						10:	(*Consigne epaisseur pour la nouvelle vitesse*)
							VAR_ParameterWriter.fbClientDataExcha.txBuffer[0]:=16#08;
							VAR_ParameterWriter.fbClientDataExcha.txBuffer[1]:=16#00;
							VAR_ParameterWriter.fbClientDataExcha.txBuffer[2]:= F_ToASC('U');
							VAR_ParameterWriter.fbClientDataExcha.txBuffer[3]:= F_ToASC('F');
							VAR_ParameterWriter.fbClientDataExcha.txBuffer[4]:= 16#0A;
							VAR_ParameterWriter.fbClientDataExcha.txBuffer[5]:= 16#01;
							MEMCPY(ADR(VAR_ParameterWriter.fbClientDataExcha.txBuffer[6]),ADR(I_Thick_SP),4);
							VAR_ParameterWriter.fbClientDataExcha.txBuffer[10] := VAR_ParameterWriter.fbClientDataExcha.txBuffer[2] +
												VAR_ParameterWriter.fbClientDataExcha.txBuffer[3] +
												VAR_ParameterWriter.fbClientDataExcha.txBuffer[4] +
												VAR_ParameterWriter.fbClientDataExcha.txBuffer[5] +
												VAR_ParameterWriter.fbClientDataExcha.txBuffer[6] +
												VAR_ParameterWriter.fbClientDataExcha.txBuffer[7] +
												VAR_ParameterWriter.fbClientDataExcha.txBuffer[8] +
												VAR_ParameterWriter.fbClientDataExcha.txBuffer[9];
							VAR_ParameterWriter.fbClientDataExcha.nbTransmittedChar := 11;
							VAR_ParameterWriter.fbClientDataExcha.nbExpectedChar := 6;


						11:	(*Nouvelle consigne de vitesse*)
							VAR_ParameterWriter.fbClientDataExcha.txBuffer[0]:=16#08;
							VAR_ParameterWriter.fbClientDataExcha.txBuffer[1]:=16#00;
							VAR_ParameterWriter.fbClientDataExcha.txBuffer[2]:= F_ToASC('U');
							VAR_ParameterWriter.fbClientDataExcha.txBuffer[3]:= F_ToASC('F');
							VAR_ParameterWriter.fbClientDataExcha.txBuffer[4]:= 16#0B;
							VAR_ParameterWriter.fbClientDataExcha.txBuffer[5]:= 16#01;
							MEMCPY(ADR(VAR_ParameterWriter.fbClientDataExcha.txBuffer[6]),ADR(I_New_Rate),4);
							VAR_ParameterWriter.fbClientDataExcha.txBuffer[10] := VAR_ParameterWriter.fbClientDataExcha.txBuffer[2] +
												VAR_ParameterWriter.fbClientDataExcha.txBuffer[3] +
												VAR_ParameterWriter.fbClientDataExcha.txBuffer[4] +
												VAR_ParameterWriter.fbClientDataExcha.txBuffer[5] +
												VAR_ParameterWriter.fbClientDataExcha.txBuffer[6] +
												VAR_ParameterWriter.fbClientDataExcha.txBuffer[7] +
												VAR_ParameterWriter.fbClientDataExcha.txBuffer[8] +
												VAR_ParameterWriter.fbClientDataExcha.txBuffer[9];
							VAR_ParameterWriter.fbClientDataExcha.nbTransmittedChar := 11;
							VAR_ParameterWriter.fbClientDataExcha.nbExpectedChar := 6;


						12:	(*Temps de monté à la nouvelle vitesse*)
							VAR_ParameterWriter.fbClientDataExcha.txBuffer[0]:=16#08;
							VAR_ParameterWriter.fbClientDataExcha.txBuffer[1]:=16#00;
							VAR_ParameterWriter.fbClientDataExcha.txBuffer[2]:= F_ToASC('U');
							VAR_ParameterWriter.fbClientDataExcha.txBuffer[3]:= F_ToASC('F');
							VAR_ParameterWriter.fbClientDataExcha.txBuffer[4]:= 16#0C;
							VAR_ParameterWriter.fbClientDataExcha.txBuffer[5]:= 16#01;
							TEMP_DWORD := UINT_TO_DWORD(I_Rate_Ramp_Time);
							MEMCPY(ADR(VAR_ParameterWriter.fbClientDataExcha.txBuffer[6]),ADR(TEMP_DWORD),4);
							VAR_ParameterWriter.fbClientDataExcha.txBuffer[10] := VAR_ParameterWriter.fbClientDataExcha.txBuffer[2] +
												VAR_ParameterWriter.fbClientDataExcha.txBuffer[3] +
												VAR_ParameterWriter.fbClientDataExcha.txBuffer[4] +
												VAR_ParameterWriter.fbClientDataExcha.txBuffer[5] +
												VAR_ParameterWriter.fbClientDataExcha.txBuffer[6] +
												VAR_ParameterWriter.fbClientDataExcha.txBuffer[7] +
												VAR_ParameterWriter.fbClientDataExcha.txBuffer[8] +
												VAR_ParameterWriter.fbClientDataExcha.txBuffer[9];
							VAR_ParameterWriter.fbClientDataExcha.nbTransmittedChar := 11;
							VAR_ParameterWriter.fbClientDataExcha.nbExpectedChar := 6;


						13:	(*Rate Watcher Accuracy*)
							VAR_ParameterWriter.fbClientDataExcha.txBuffer[0]:=16#08;
							VAR_ParameterWriter.fbClientDataExcha.txBuffer[1]:=16#00;
							VAR_ParameterWriter.fbClientDataExcha.txBuffer[2]:= F_ToASC('U');
							VAR_ParameterWriter.fbClientDataExcha.txBuffer[3]:= F_ToASC('F');
							VAR_ParameterWriter.fbClientDataExcha.txBuffer[4]:= 16#0D;
							VAR_ParameterWriter.fbClientDataExcha.txBuffer[5]:= 16#01;
							TEMP_DWORD := INT_TO_DWORD(I_Rate_Watcher_Accuracy);
							MEMCPY(ADR(VAR_ParameterWriter.fbClientDataExcha.txBuffer[6]),ADR(TEMP_DWORD),4);
							VAR_ParameterWriter.fbClientDataExcha.txBuffer[10] := VAR_ParameterWriter.fbClientDataExcha.txBuffer[2] +
												VAR_ParameterWriter.fbClientDataExcha.txBuffer[3] +
												VAR_ParameterWriter.fbClientDataExcha.txBuffer[4] +
												VAR_ParameterWriter.fbClientDataExcha.txBuffer[5] +
												VAR_ParameterWriter.fbClientDataExcha.txBuffer[6] +
												VAR_ParameterWriter.fbClientDataExcha.txBuffer[7] +
												VAR_ParameterWriter.fbClientDataExcha.txBuffer[8] +
												VAR_ParameterWriter.fbClientDataExcha.txBuffer[9];
							VAR_ParameterWriter.fbClientDataExcha.nbTransmittedChar := 11;
							VAR_ParameterWriter.fbClientDataExcha.nbExpectedChar := 6;


						14:	(*RW hold time*)
							VAR_ParameterWriter.fbClientDataExcha.txBuffer[0]:=16#08;
							VAR_ParameterWriter.fbClientDataExcha.txBuffer[1]:=16#00;
							VAR_ParameterWriter.fbClientDataExcha.txBuffer[2]:= F_ToASC('U');
							VAR_ParameterWriter.fbClientDataExcha.txBuffer[3]:= F_ToASC('F');
							VAR_ParameterWriter.fbClientDataExcha.txBuffer[4]:= 16#0E;
							VAR_ParameterWriter.fbClientDataExcha.txBuffer[5]:= 16#01;
							TEMP_DWORD := INT_TO_DWORD(I_RW_Hold_Time);
							MEMCPY(ADR(VAR_ParameterWriter.fbClientDataExcha.txBuffer[6]),ADR(TEMP_DWORD),4);
							VAR_ParameterWriter.fbClientDataExcha.txBuffer[10] := VAR_ParameterWriter.fbClientDataExcha.txBuffer[2] +
												VAR_ParameterWriter.fbClientDataExcha.txBuffer[3] +
												VAR_ParameterWriter.fbClientDataExcha.txBuffer[4] +
												VAR_ParameterWriter.fbClientDataExcha.txBuffer[5] +
												VAR_ParameterWriter.fbClientDataExcha.txBuffer[6] +
												VAR_ParameterWriter.fbClientDataExcha.txBuffer[7] +
												VAR_ParameterWriter.fbClientDataExcha.txBuffer[8] +
												VAR_ParameterWriter.fbClientDataExcha.txBuffer[9];
							VAR_ParameterWriter.fbClientDataExcha.nbTransmittedChar := 11;
							VAR_ParameterWriter.fbClientDataExcha.nbExpectedChar := 6;


						15:	(*Sensor à utiliser*)
							VAR_ParameterWriter.fbClientDataExcha.txBuffer[0]:=16#08;
							VAR_ParameterWriter.fbClientDataExcha.txBuffer[1]:=16#00;
							VAR_ParameterWriter.fbClientDataExcha.txBuffer[2]:= F_ToASC('U');
							VAR_ParameterWriter.fbClientDataExcha.txBuffer[3]:= F_ToASC('F');
							VAR_ParameterWriter.fbClientDataExcha.txBuffer[4]:= 16#0F;
							VAR_ParameterWriter.fbClientDataExcha.txBuffer[5]:= 16#01;
							TEMP_DWORD := BYTE_TO_DWORD(I_Sensor);
							MEMCPY(ADR(VAR_ParameterWriter.fbClientDataExcha.txBuffer[6]),ADR(TEMP_DWORD),4);
							VAR_ParameterWriter.fbClientDataExcha.txBuffer[10] := VAR_ParameterWriter.fbClientDataExcha.txBuffer[2] +
												VAR_ParameterWriter.fbClientDataExcha.txBuffer[3] +
												VAR_ParameterWriter.fbClientDataExcha.txBuffer[4] +
												VAR_ParameterWriter.fbClientDataExcha.txBuffer[5] +
												VAR_ParameterWriter.fbClientDataExcha.txBuffer[6] +
												VAR_ParameterWriter.fbClientDataExcha.txBuffer[7] +
												VAR_ParameterWriter.fbClientDataExcha.txBuffer[8] +
												VAR_ParameterWriter.fbClientDataExcha.txBuffer[9];
							VAR_ParameterWriter.fbClientDataExcha.nbTransmittedChar := 11;
							VAR_ParameterWriter.fbClientDataExcha.nbExpectedChar := 6;


						16:	(*Facteur de correction 1*)
							VAR_ParameterWriter.fbClientDataExcha.txBuffer[0]:=16#08;
							VAR_ParameterWriter.fbClientDataExcha.txBuffer[1]:=16#00;
							VAR_ParameterWriter.fbClientDataExcha.txBuffer[2]:= F_ToASC('U');
							VAR_ParameterWriter.fbClientDataExcha.txBuffer[3]:= F_ToASC('F');
							VAR_ParameterWriter.fbClientDataExcha.txBuffer[4]:= 16#10;
							VAR_ParameterWriter.fbClientDataExcha.txBuffer[5]:= 16#01;
							MEMCPY(ADR(VAR_ParameterWriter.fbClientDataExcha.txBuffer[6]),ADR(I_Tool_Factor1),4);
							VAR_ParameterWriter.fbClientDataExcha.txBuffer[10] := VAR_ParameterWriter.fbClientDataExcha.txBuffer[2] +
												VAR_ParameterWriter.fbClientDataExcha.txBuffer[3] +
												VAR_ParameterWriter.fbClientDataExcha.txBuffer[4] +
												VAR_ParameterWriter.fbClientDataExcha.txBuffer[5] +
												VAR_ParameterWriter.fbClientDataExcha.txBuffer[6] +
												VAR_ParameterWriter.fbClientDataExcha.txBuffer[7] +
												VAR_ParameterWriter.fbClientDataExcha.txBuffer[8] +
												VAR_ParameterWriter.fbClientDataExcha.txBuffer[9];
							VAR_ParameterWriter.fbClientDataExcha.nbTransmittedChar := 11;
							VAR_ParameterWriter.fbClientDataExcha.nbExpectedChar := 6;



						17:	(*Facteur de correction 2*)
							VAR_ParameterWriter.fbClientDataExcha.txBuffer[0]:=16#08;
							VAR_ParameterWriter.fbClientDataExcha.txBuffer[1]:=16#00;
							VAR_ParameterWriter.fbClientDataExcha.txBuffer[2]:= F_ToASC('U');
							VAR_ParameterWriter.fbClientDataExcha.txBuffer[3]:= F_ToASC('F');
							VAR_ParameterWriter.fbClientDataExcha.txBuffer[4]:= 16#11;
							VAR_ParameterWriter.fbClientDataExcha.txBuffer[5]:= 16#01;
							MEMCPY(ADR(VAR_ParameterWriter.fbClientDataExcha.txBuffer[6]),ADR(I_Tool_Factor2),4);
							VAR_ParameterWriter.fbClientDataExcha.txBuffer[10] := VAR_ParameterWriter.fbClientDataExcha.txBuffer[2] +
												VAR_ParameterWriter.fbClientDataExcha.txBuffer[3] +
												VAR_ParameterWriter.fbClientDataExcha.txBuffer[4] +
												VAR_ParameterWriter.fbClientDataExcha.txBuffer[5] +
												VAR_ParameterWriter.fbClientDataExcha.txBuffer[6] +
												VAR_ParameterWriter.fbClientDataExcha.txBuffer[7] +
												VAR_ParameterWriter.fbClientDataExcha.txBuffer[8] +
												VAR_ParameterWriter.fbClientDataExcha.txBuffer[9];
							VAR_ParameterWriter.fbClientDataExcha.nbTransmittedChar := 11;
							VAR_ParameterWriter.fbClientDataExcha.nbExpectedChar := 6;



						18:	(*Xtal stabilility single*)
							VAR_ParameterWriter.fbClientDataExcha.txBuffer[0]:=16#08;
							VAR_ParameterWriter.fbClientDataExcha.txBuffer[1]:=16#00;
							VAR_ParameterWriter.fbClientDataExcha.txBuffer[2]:= F_ToASC('U');
							VAR_ParameterWriter.fbClientDataExcha.txBuffer[3]:= F_ToASC('F');
							VAR_ParameterWriter.fbClientDataExcha.txBuffer[4]:= 16#12;
							VAR_ParameterWriter.fbClientDataExcha.txBuffer[5]:= 16#01;
							TEMP_DWORD := UINT_TO_DWORD(I_Stab_Single);
							MEMCPY(ADR(VAR_ParameterWriter.fbClientDataExcha.txBuffer[6]),ADR(TEMP_DWORD),4);
							VAR_ParameterWriter.fbClientDataExcha.txBuffer[10] := VAR_ParameterWriter.fbClientDataExcha.txBuffer[2] +
												VAR_ParameterWriter.fbClientDataExcha.txBuffer[3] +
												VAR_ParameterWriter.fbClientDataExcha.txBuffer[4] +
												VAR_ParameterWriter.fbClientDataExcha.txBuffer[5] +
												VAR_ParameterWriter.fbClientDataExcha.txBuffer[6] +
												VAR_ParameterWriter.fbClientDataExcha.txBuffer[7] +
												VAR_ParameterWriter.fbClientDataExcha.txBuffer[8] +
												VAR_ParameterWriter.fbClientDataExcha.txBuffer[9];
							VAR_ParameterWriter.fbClientDataExcha.nbTransmittedChar := 11;
							VAR_ParameterWriter.fbClientDataExcha.nbExpectedChar := 6;


						19:	(*Xtal stabilility total*)
							VAR_ParameterWriter.fbClientDataExcha.txBuffer[0]:=16#08;
							VAR_ParameterWriter.fbClientDataExcha.txBuffer[1]:=16#00;
							VAR_ParameterWriter.fbClientDataExcha.txBuffer[2]:= F_ToASC('U');
							VAR_ParameterWriter.fbClientDataExcha.txBuffer[3]:= F_ToASC('F');
							VAR_ParameterWriter.fbClientDataExcha.txBuffer[4]:= 16#13;
							VAR_ParameterWriter.fbClientDataExcha.txBuffer[5]:= 16#01;
							TEMP_DWORD := UINT_TO_DWORD(I_Stab_Total);
							MEMCPY(ADR(VAR_ParameterWriter.fbClientDataExcha.txBuffer[6]),ADR(TEMP_DWORD),4);
							VAR_ParameterWriter.fbClientDataExcha.txBuffer[10] := VAR_ParameterWriter.fbClientDataExcha.txBuffer[2] +
												VAR_ParameterWriter.fbClientDataExcha.txBuffer[3] +
												VAR_ParameterWriter.fbClientDataExcha.txBuffer[4] +
												VAR_ParameterWriter.fbClientDataExcha.txBuffer[5] +
												VAR_ParameterWriter.fbClientDataExcha.txBuffer[6] +
												VAR_ParameterWriter.fbClientDataExcha.txBuffer[7] +
												VAR_ParameterWriter.fbClientDataExcha.txBuffer[8] +
												VAR_ParameterWriter.fbClientDataExcha.txBuffer[9];
							VAR_ParameterWriter.fbClientDataExcha.nbTransmittedChar := 11;
							VAR_ParameterWriter.fbClientDataExcha.nbExpectedChar := 6;


						20:	(*Xtal quality percent*)
							VAR_ParameterWriter.fbClientDataExcha.txBuffer[0]:=16#08;
							VAR_ParameterWriter.fbClientDataExcha.txBuffer[1]:=16#00;
							VAR_ParameterWriter.fbClientDataExcha.txBuffer[2]:= F_ToASC('U');
							VAR_ParameterWriter.fbClientDataExcha.txBuffer[3]:= F_ToASC('F');
							VAR_ParameterWriter.fbClientDataExcha.txBuffer[4]:= 16#14;
							VAR_ParameterWriter.fbClientDataExcha.txBuffer[5]:= 16#01;
							TEMP_DWORD := USINT_TO_DWORD(I_Quality_percent);
							MEMCPY(ADR(VAR_ParameterWriter.fbClientDataExcha.txBuffer[6]),ADR(TEMP_DWORD),4);
							VAR_ParameterWriter.fbClientDataExcha.txBuffer[10] := VAR_ParameterWriter.fbClientDataExcha.txBuffer[2] +
												VAR_ParameterWriter.fbClientDataExcha.txBuffer[3] +
												VAR_ParameterWriter.fbClientDataExcha.txBuffer[4] +
												VAR_ParameterWriter.fbClientDataExcha.txBuffer[5] +
												VAR_ParameterWriter.fbClientDataExcha.txBuffer[6] +
												VAR_ParameterWriter.fbClientDataExcha.txBuffer[7] +
												VAR_ParameterWriter.fbClientDataExcha.txBuffer[8] +
												VAR_ParameterWriter.fbClientDataExcha.txBuffer[9];
							VAR_ParameterWriter.fbClientDataExcha.nbTransmittedChar := 11;
							VAR_ParameterWriter.fbClientDataExcha.nbExpectedChar := 6;


						21:	(*Xtal quality Counts*)
							VAR_ParameterWriter.fbClientDataExcha.txBuffer[0]:=16#08;
							VAR_ParameterWriter.fbClientDataExcha.txBuffer[1]:=16#00;
							VAR_ParameterWriter.fbClientDataExcha.txBuffer[2]:= F_ToASC('U');
							VAR_ParameterWriter.fbClientDataExcha.txBuffer[3]:= F_ToASC('F');
							VAR_ParameterWriter.fbClientDataExcha.txBuffer[4]:= 16#15;
							VAR_ParameterWriter.fbClientDataExcha.txBuffer[5]:= 16#01;
							TEMP_DWORD := USINT_TO_DWORD(I_Quality_Counts);
							MEMCPY(ADR(VAR_ParameterWriter.fbClientDataExcha.txBuffer[6]),ADR(TEMP_DWORD),4);
							VAR_ParameterWriter.fbClientDataExcha.txBuffer[10] := VAR_ParameterWriter.fbClientDataExcha.txBuffer[2] +
												VAR_ParameterWriter.fbClientDataExcha.txBuffer[3] +
												VAR_ParameterWriter.fbClientDataExcha.txBuffer[4] +
												VAR_ParameterWriter.fbClientDataExcha.txBuffer[5] +
												VAR_ParameterWriter.fbClientDataExcha.txBuffer[6] +
												VAR_ParameterWriter.fbClientDataExcha.txBuffer[7] +
												VAR_ParameterWriter.fbClientDataExcha.txBuffer[8] +
												VAR_ParameterWriter.fbClientDataExcha.txBuffer[9];
							VAR_ParameterWriter.fbClientDataExcha.nbTransmittedChar := 11;
							VAR_ParameterWriter.fbClientDataExcha.nbExpectedChar := 6;


						22:	(*Source*)
							VAR_ParameterWriter.fbClientDataExcha.txBuffer[0]:=16#08;
							VAR_ParameterWriter.fbClientDataExcha.txBuffer[1]:=16#00;
							VAR_ParameterWriter.fbClientDataExcha.txBuffer[2]:= F_ToASC('U');
							VAR_ParameterWriter.fbClientDataExcha.txBuffer[3]:= F_ToASC('F');
							VAR_ParameterWriter.fbClientDataExcha.txBuffer[4]:= 16#16;
							VAR_ParameterWriter.fbClientDataExcha.txBuffer[5]:= 16#01;
							TEMP_DWORD := BYTE_TO_DWORD(I_Source);
							MEMCPY(ADR(VAR_ParameterWriter.fbClientDataExcha.txBuffer[6]),ADR(TEMP_DWORD),4);
							VAR_ParameterWriter.fbClientDataExcha.txBuffer[10] := VAR_ParameterWriter.fbClientDataExcha.txBuffer[2] +
												VAR_ParameterWriter.fbClientDataExcha.txBuffer[3] +
												VAR_ParameterWriter.fbClientDataExcha.txBuffer[4] +
												VAR_ParameterWriter.fbClientDataExcha.txBuffer[5] +
												VAR_ParameterWriter.fbClientDataExcha.txBuffer[6] +
												VAR_ParameterWriter.fbClientDataExcha.txBuffer[7] +
												VAR_ParameterWriter.fbClientDataExcha.txBuffer[8] +
												VAR_ParameterWriter.fbClientDataExcha.txBuffer[9];
							VAR_ParameterWriter.fbClientDataExcha.nbTransmittedChar := 11;
							VAR_ParameterWriter.fbClientDataExcha.nbExpectedChar := 6;


						23:	(*Source*)
							VAR_ParameterWriter.fbClientDataExcha.txBuffer[0]:=16#08;
							VAR_ParameterWriter.fbClientDataExcha.txBuffer[1]:=16#00;
							VAR_ParameterWriter.fbClientDataExcha.txBuffer[2]:= F_ToASC('U');
							VAR_ParameterWriter.fbClientDataExcha.txBuffer[3]:= F_ToASC('F');
							VAR_ParameterWriter.fbClientDataExcha.txBuffer[4]:= 16#17;
							VAR_ParameterWriter.fbClientDataExcha.txBuffer[5]:= 16#01;
							TEMP_DWORD := BYTE_TO_DWORD(I_Crucible_Nb);
							MEMCPY(ADR(VAR_ParameterWriter.fbClientDataExcha.txBuffer[6]),ADR(TEMP_DWORD),4);
							VAR_ParameterWriter.fbClientDataExcha.txBuffer[10] := VAR_ParameterWriter.fbClientDataExcha.txBuffer[2] +
												VAR_ParameterWriter.fbClientDataExcha.txBuffer[3] +
												VAR_ParameterWriter.fbClientDataExcha.txBuffer[4] +
												VAR_ParameterWriter.fbClientDataExcha.txBuffer[5] +
												VAR_ParameterWriter.fbClientDataExcha.txBuffer[6] +
												VAR_ParameterWriter.fbClientDataExcha.txBuffer[7] +
												VAR_ParameterWriter.fbClientDataExcha.txBuffer[8] +
												VAR_ParameterWriter.fbClientDataExcha.txBuffer[9];
							VAR_ParameterWriter.fbClientDataExcha.nbTransmittedChar := 11;
							VAR_ParameterWriter.fbClientDataExcha.nbExpectedChar := 6;


						24:	(*PID Gain*)
							VAR_ParameterWriter.fbClientDataExcha.txBuffer[0]:=16#08;
							VAR_ParameterWriter.fbClientDataExcha.txBuffer[1]:=16#00;
							VAR_ParameterWriter.fbClientDataExcha.txBuffer[2]:= F_ToASC('U');
							VAR_ParameterWriter.fbClientDataExcha.txBuffer[3]:= F_ToASC('F');
							VAR_ParameterWriter.fbClientDataExcha.txBuffer[4]:= 16#18;
							VAR_ParameterWriter.fbClientDataExcha.txBuffer[5]:= 16#01;
							MEMCPY(ADR(VAR_ParameterWriter.fbClientDataExcha.txBuffer[6]),ADR(I_PID_GAIN),4);
							VAR_ParameterWriter.fbClientDataExcha.txBuffer[10] := VAR_ParameterWriter.fbClientDataExcha.txBuffer[2] +
												VAR_ParameterWriter.fbClientDataExcha.txBuffer[3] +
												VAR_ParameterWriter.fbClientDataExcha.txBuffer[4] +
												VAR_ParameterWriter.fbClientDataExcha.txBuffer[5] +
												VAR_ParameterWriter.fbClientDataExcha.txBuffer[6] +
												VAR_ParameterWriter.fbClientDataExcha.txBuffer[7] +
												VAR_ParameterWriter.fbClientDataExcha.txBuffer[8] +
												VAR_ParameterWriter.fbClientDataExcha.txBuffer[9];
							VAR_ParameterWriter.fbClientDataExcha.nbTransmittedChar := 11;
							VAR_ParameterWriter.fbClientDataExcha.nbExpectedChar := 6;


						25:	(*PID Integral - control time constant*)
							VAR_ParameterWriter.fbClientDataExcha.txBuffer[0]:=16#08;
							VAR_ParameterWriter.fbClientDataExcha.txBuffer[1]:=16#00;
							VAR_ParameterWriter.fbClientDataExcha.txBuffer[2]:= F_ToASC('U');
							VAR_ParameterWriter.fbClientDataExcha.txBuffer[3]:= F_ToASC('F');
							VAR_ParameterWriter.fbClientDataExcha.txBuffer[4]:= 16#19;
							VAR_ParameterWriter.fbClientDataExcha.txBuffer[5]:= 16#01;
							MEMCPY(ADR(VAR_ParameterWriter.fbClientDataExcha.txBuffer[6]),ADR(I_PID_Ti),4);
							VAR_ParameterWriter.fbClientDataExcha.txBuffer[10] := VAR_ParameterWriter.fbClientDataExcha.txBuffer[2] +
												VAR_ParameterWriter.fbClientDataExcha.txBuffer[3] +
												VAR_ParameterWriter.fbClientDataExcha.txBuffer[4] +
												VAR_ParameterWriter.fbClientDataExcha.txBuffer[5] +
												VAR_ParameterWriter.fbClientDataExcha.txBuffer[6] +
												VAR_ParameterWriter.fbClientDataExcha.txBuffer[7] +
												VAR_ParameterWriter.fbClientDataExcha.txBuffer[8] +
												VAR_ParameterWriter.fbClientDataExcha.txBuffer[9];
							VAR_ParameterWriter.fbClientDataExcha.nbTransmittedChar := 11;
							VAR_ParameterWriter.fbClientDataExcha.nbExpectedChar := 6;


						26:	(*PID Dérivée - control dead time*)
							VAR_ParameterWriter.fbClientDataExcha.txBuffer[0]:=16#08;
							VAR_ParameterWriter.fbClientDataExcha.txBuffer[1]:=16#00;
							VAR_ParameterWriter.fbClientDataExcha.txBuffer[2]:= F_ToASC('U');
							VAR_ParameterWriter.fbClientDataExcha.txBuffer[3]:= F_ToASC('F');
							VAR_ParameterWriter.fbClientDataExcha.txBuffer[4]:= 16#1A;
							VAR_ParameterWriter.fbClientDataExcha.txBuffer[5]:= 16#01;
							MEMCPY(ADR(VAR_ParameterWriter.fbClientDataExcha.txBuffer[6]),ADR(I_PID_Td),4);
							VAR_ParameterWriter.fbClientDataExcha.txBuffer[10] := VAR_ParameterWriter.fbClientDataExcha.txBuffer[2] +
												VAR_ParameterWriter.fbClientDataExcha.txBuffer[3] +
												VAR_ParameterWriter.fbClientDataExcha.txBuffer[4] +
												VAR_ParameterWriter.fbClientDataExcha.txBuffer[5] +
												VAR_ParameterWriter.fbClientDataExcha.txBuffer[6] +
												VAR_ParameterWriter.fbClientDataExcha.txBuffer[7] +
												VAR_ParameterWriter.fbClientDataExcha.txBuffer[8] +
												VAR_ParameterWriter.fbClientDataExcha.txBuffer[9];
							VAR_ParameterWriter.fbClientDataExcha.nbTransmittedChar := 11;
							VAR_ParameterWriter.fbClientDataExcha.nbExpectedChar := 6;


						27:	(*Max Power*)
							VAR_ParameterWriter.fbClientDataExcha.txBuffer[0]:=16#08;
							VAR_ParameterWriter.fbClientDataExcha.txBuffer[1]:=16#00;
							VAR_ParameterWriter.fbClientDataExcha.txBuffer[2]:= F_ToASC('U');
							VAR_ParameterWriter.fbClientDataExcha.txBuffer[3]:= F_ToASC('F');
							VAR_ParameterWriter.fbClientDataExcha.txBuffer[4]:= 16#1B;
							VAR_ParameterWriter.fbClientDataExcha.txBuffer[5]:= 16#01;
							MEMCPY(ADR(VAR_ParameterWriter.fbClientDataExcha.txBuffer[6]),ADR(I_Max_Power),4);
							VAR_ParameterWriter.fbClientDataExcha.txBuffer[10] := VAR_ParameterWriter.fbClientDataExcha.txBuffer[2] +
												VAR_ParameterWriter.fbClientDataExcha.txBuffer[3] +
												VAR_ParameterWriter.fbClientDataExcha.txBuffer[4] +
												VAR_ParameterWriter.fbClientDataExcha.txBuffer[5] +
												VAR_ParameterWriter.fbClientDataExcha.txBuffer[6] +
												VAR_ParameterWriter.fbClientDataExcha.txBuffer[7] +
												VAR_ParameterWriter.fbClientDataExcha.txBuffer[8] +
												VAR_ParameterWriter.fbClientDataExcha.txBuffer[9];
							VAR_ParameterWriter.fbClientDataExcha.nbTransmittedChar := 11;
							VAR_ParameterWriter.fbClientDataExcha.nbExpectedChar := 6;


						28:	(*Densité*)
							VAR_ParameterWriter.fbClientDataExcha.txBuffer[0]:=16#08;
							VAR_ParameterWriter.fbClientDataExcha.txBuffer[1]:=16#00;
							VAR_ParameterWriter.fbClientDataExcha.txBuffer[2]:= F_ToASC('U');
							VAR_ParameterWriter.fbClientDataExcha.txBuffer[3]:= F_ToASC('F');
							VAR_ParameterWriter.fbClientDataExcha.txBuffer[4]:= 16#1C;
							VAR_ParameterWriter.fbClientDataExcha.txBuffer[5]:= 16#01;
							MEMCPY(ADR(VAR_ParameterWriter.fbClientDataExcha.txBuffer[6]),ADR(I_Densite),4);
							VAR_ParameterWriter.fbClientDataExcha.txBuffer[10] := VAR_ParameterWriter.fbClientDataExcha.txBuffer[2] +
												VAR_ParameterWriter.fbClientDataExcha.txBuffer[3] +
												VAR_ParameterWriter.fbClientDataExcha.txBuffer[4] +
												VAR_ParameterWriter.fbClientDataExcha.txBuffer[5] +
												VAR_ParameterWriter.fbClientDataExcha.txBuffer[6] +
												VAR_ParameterWriter.fbClientDataExcha.txBuffer[7] +
												VAR_ParameterWriter.fbClientDataExcha.txBuffer[8] +
												VAR_ParameterWriter.fbClientDataExcha.txBuffer[9];
							VAR_ParameterWriter.fbClientDataExcha.nbTransmittedChar := 11;
							VAR_ParameterWriter.fbClientDataExcha.nbExpectedChar := 6;

						29:	(*Z-Ratio*)
							VAR_ParameterWriter.fbClientDataExcha.txBuffer[0]:=16#08;
							VAR_ParameterWriter.fbClientDataExcha.txBuffer[1]:=16#00;
							VAR_ParameterWriter.fbClientDataExcha.txBuffer[2]:= F_ToASC('U');
							VAR_ParameterWriter.fbClientDataExcha.txBuffer[3]:= F_ToASC('F');
							VAR_ParameterWriter.fbClientDataExcha.txBuffer[4]:= 16#1D;
							VAR_ParameterWriter.fbClientDataExcha.txBuffer[5]:= 16#01;
							MEMCPY(ADR(VAR_ParameterWriter.fbClientDataExcha.txBuffer[6]),ADR(I_ZRatio),4);
							VAR_ParameterWriter.fbClientDataExcha.txBuffer[10] := VAR_ParameterWriter.fbClientDataExcha.txBuffer[2] +
												VAR_ParameterWriter.fbClientDataExcha.txBuffer[3] +
												VAR_ParameterWriter.fbClientDataExcha.txBuffer[4] +
												VAR_ParameterWriter.fbClientDataExcha.txBuffer[5] +
												VAR_ParameterWriter.fbClientDataExcha.txBuffer[6] +
												VAR_ParameterWriter.fbClientDataExcha.txBuffer[7] +
												VAR_ParameterWriter.fbClientDataExcha.txBuffer[8] +
												VAR_ParameterWriter.fbClientDataExcha.txBuffer[9];
							VAR_ParameterWriter.fbClientDataExcha.nbTransmittedChar := 11;
							VAR_ParameterWriter.fbClientDataExcha.nbExpectedChar := 6;

						30:	(*TimePower*)
							VAR_ParameterWriter.fbClientDataExcha.txBuffer[0]:=16#08;
							VAR_ParameterWriter.fbClientDataExcha.txBuffer[1]:=16#00;
							VAR_ParameterWriter.fbClientDataExcha.txBuffer[2]:= F_ToASC('U');
							VAR_ParameterWriter.fbClientDataExcha.txBuffer[3]:= F_ToASC('F');
							VAR_ParameterWriter.fbClientDataExcha.txBuffer[4]:= 16#1E;
							VAR_ParameterWriter.fbClientDataExcha.txBuffer[5]:= 16#01;
							TEMP_DWORD := BOOL_TO_DWORD(I_TIME_POWER);
							MEMCPY(ADR(VAR_ParameterWriter.fbClientDataExcha.txBuffer[6]),ADR(TEMP_DWORD),4);
							VAR_ParameterWriter.fbClientDataExcha.txBuffer[10] := VAR_ParameterWriter.fbClientDataExcha.txBuffer[2] +
												VAR_ParameterWriter.fbClientDataExcha.txBuffer[3] +
												VAR_ParameterWriter.fbClientDataExcha.txBuffer[4] +
												VAR_ParameterWriter.fbClientDataExcha.txBuffer[5] +
												VAR_ParameterWriter.fbClientDataExcha.txBuffer[6] +
												VAR_ParameterWriter.fbClientDataExcha.txBuffer[7] +
												VAR_ParameterWriter.fbClientDataExcha.txBuffer[8] +
												VAR_ParameterWriter.fbClientDataExcha.txBuffer[9];
							VAR_ParameterWriter.fbClientDataExcha.nbTransmittedChar := 11;
							VAR_ParameterWriter.fbClientDataExcha.nbExpectedChar := 6;

						31:	(*Delay Option*)
							VAR_ParameterWriter.fbClientDataExcha.txBuffer[0]:=16#08;
							VAR_ParameterWriter.fbClientDataExcha.txBuffer[1]:=16#00;
							VAR_ParameterWriter.fbClientDataExcha.txBuffer[2]:= F_ToASC('U');
							VAR_ParameterWriter.fbClientDataExcha.txBuffer[3]:= F_ToASC('F');
							VAR_ParameterWriter.fbClientDataExcha.txBuffer[4]:= 16#1F;
							VAR_ParameterWriter.fbClientDataExcha.txBuffer[5]:= 16#01;
							TEMP_DWORD := BYTE_TO_DWORD(I_Delay_Option);
							MEMCPY(ADR(VAR_ParameterWriter.fbClientDataExcha.txBuffer[6]),ADR(TEMP_DWORD),4);
							VAR_ParameterWriter.fbClientDataExcha.txBuffer[10] := VAR_ParameterWriter.fbClientDataExcha.txBuffer[2] +
												VAR_ParameterWriter.fbClientDataExcha.txBuffer[3] +
												VAR_ParameterWriter.fbClientDataExcha.txBuffer[4] +
												VAR_ParameterWriter.fbClientDataExcha.txBuffer[5] +
												VAR_ParameterWriter.fbClientDataExcha.txBuffer[6] +
												VAR_ParameterWriter.fbClientDataExcha.txBuffer[7] +
												VAR_ParameterWriter.fbClientDataExcha.txBuffer[8] +
												VAR_ParameterWriter.fbClientDataExcha.txBuffer[9];
							VAR_ParameterWriter.fbClientDataExcha.nbTransmittedChar := 11;
							VAR_ParameterWriter.fbClientDataExcha.nbExpectedChar := 6;

						32:	(*Transfer Sensor*)
							VAR_ParameterWriter.fbClientDataExcha.txBuffer[0]:=16#08;
							VAR_ParameterWriter.fbClientDataExcha.txBuffer[1]:=16#00;
							VAR_ParameterWriter.fbClientDataExcha.txBuffer[2]:= F_ToASC('U');
							VAR_ParameterWriter.fbClientDataExcha.txBuffer[3]:= F_ToASC('F');
							VAR_ParameterWriter.fbClientDataExcha.txBuffer[4]:= 16#20;
							VAR_ParameterWriter.fbClientDataExcha.txBuffer[5]:= 16#01;
							TEMP_DWORD := INT_TO_DWORD(I_Transfer_sensor);
							MEMCPY(ADR(VAR_ParameterWriter.fbClientDataExcha.txBuffer[6]),ADR(TEMP_DWORD),4);
							VAR_ParameterWriter.fbClientDataExcha.txBuffer[10] := VAR_ParameterWriter.fbClientDataExcha.txBuffer[2] +
												VAR_ParameterWriter.fbClientDataExcha.txBuffer[3] +
												VAR_ParameterWriter.fbClientDataExcha.txBuffer[4] +
												VAR_ParameterWriter.fbClientDataExcha.txBuffer[5] +
												VAR_ParameterWriter.fbClientDataExcha.txBuffer[6] +
												VAR_ParameterWriter.fbClientDataExcha.txBuffer[7] +
												VAR_ParameterWriter.fbClientDataExcha.txBuffer[8] +
												VAR_ParameterWriter.fbClientDataExcha.txBuffer[9];
							VAR_ParameterWriter.fbClientDataExcha.nbTransmittedChar := 11;
							VAR_ParameterWriter.fbClientDataExcha.nbExpectedChar := 6;

						33:	(*Transfer Tooling*)
							VAR_ParameterWriter.fbClientDataExcha.txBuffer[0]:=16#08;
							VAR_ParameterWriter.fbClientDataExcha.txBuffer[1]:=16#00;
							VAR_ParameterWriter.fbClientDataExcha.txBuffer[2]:= F_ToASC('U');
							VAR_ParameterWriter.fbClientDataExcha.txBuffer[3]:= F_ToASC('F');
							VAR_ParameterWriter.fbClientDataExcha.txBuffer[4]:= 16#21;
							VAR_ParameterWriter.fbClientDataExcha.txBuffer[5]:= 16#01;
							MEMCPY(ADR(VAR_ParameterWriter.fbClientDataExcha.txBuffer[6]),ADR(I_Transfer_Tool),4);
							VAR_ParameterWriter.fbClientDataExcha.txBuffer[10] := VAR_ParameterWriter.fbClientDataExcha.txBuffer[2] +
												VAR_ParameterWriter.fbClientDataExcha.txBuffer[3] +
												VAR_ParameterWriter.fbClientDataExcha.txBuffer[4] +
												VAR_ParameterWriter.fbClientDataExcha.txBuffer[5] +
												VAR_ParameterWriter.fbClientDataExcha.txBuffer[6] +
												VAR_ParameterWriter.fbClientDataExcha.txBuffer[7] +
												VAR_ParameterWriter.fbClientDataExcha.txBuffer[8] +
												VAR_ParameterWriter.fbClientDataExcha.txBuffer[9];
							VAR_ParameterWriter.fbClientDataExcha.nbTransmittedChar := 11;
							VAR_ParameterWriter.fbClientDataExcha.nbExpectedChar := 6;

						34:	(*Control Delay Time*)
							VAR_ParameterWriter.fbClientDataExcha.txBuffer[0]:=16#08;
							VAR_ParameterWriter.fbClientDataExcha.txBuffer[1]:=16#00;
							VAR_ParameterWriter.fbClientDataExcha.txBuffer[2]:= F_ToASC('U');
							VAR_ParameterWriter.fbClientDataExcha.txBuffer[3]:= F_ToASC('F');
							VAR_ParameterWriter.fbClientDataExcha.txBuffer[4]:= 16#22;
							VAR_ParameterWriter.fbClientDataExcha.txBuffer[5]:= 16#01;
							TEMP_DWORD := INT_TO_DWORD(I_Ctrl_Delay_Time);
							MEMCPY(ADR(VAR_ParameterWriter.fbClientDataExcha.txBuffer[6]),ADR(TEMP_DWORD),4);
							VAR_ParameterWriter.fbClientDataExcha.txBuffer[10] := VAR_ParameterWriter.fbClientDataExcha.txBuffer[2] +
												VAR_ParameterWriter.fbClientDataExcha.txBuffer[3] +
												VAR_ParameterWriter.fbClientDataExcha.txBuffer[4] +
												VAR_ParameterWriter.fbClientDataExcha.txBuffer[5] +
												VAR_ParameterWriter.fbClientDataExcha.txBuffer[6] +
												VAR_ParameterWriter.fbClientDataExcha.txBuffer[7] +
												VAR_ParameterWriter.fbClientDataExcha.txBuffer[8] +
												VAR_ParameterWriter.fbClientDataExcha.txBuffer[9];
							VAR_ParameterWriter.fbClientDataExcha.nbTransmittedChar := 11;
							VAR_ParameterWriter.fbClientDataExcha.nbExpectedChar := 6;

						35:	(*Ion assisted deposition*)
							VAR_ParameterWriter.fbClientDataExcha.txBuffer[0]:=16#08;
							VAR_ParameterWriter.fbClientDataExcha.txBuffer[1]:=16#00;
							VAR_ParameterWriter.fbClientDataExcha.txBuffer[2]:= F_ToASC('U');
							VAR_ParameterWriter.fbClientDataExcha.txBuffer[3]:= F_ToASC('F');
							VAR_ParameterWriter.fbClientDataExcha.txBuffer[4]:= 16#23;
							VAR_ParameterWriter.fbClientDataExcha.txBuffer[5]:= 16#01;
							TEMP_DWORD := BOOL_TO_DWORD(I_IAD_DEPOSIT);
							MEMCPY(ADR(VAR_ParameterWriter.fbClientDataExcha.txBuffer[6]),ADR(TEMP_DWORD),4);
							VAR_ParameterWriter.fbClientDataExcha.txBuffer[10] := VAR_ParameterWriter.fbClientDataExcha.txBuffer[2] +
												VAR_ParameterWriter.fbClientDataExcha.txBuffer[3] +
												VAR_ParameterWriter.fbClientDataExcha.txBuffer[4] +
												VAR_ParameterWriter.fbClientDataExcha.txBuffer[5] +
												VAR_ParameterWriter.fbClientDataExcha.txBuffer[6] +
												VAR_ParameterWriter.fbClientDataExcha.txBuffer[7] +
												VAR_ParameterWriter.fbClientDataExcha.txBuffer[8] +
												VAR_ParameterWriter.fbClientDataExcha.txBuffer[9];
							VAR_ParameterWriter.fbClientDataExcha.nbTransmittedChar := 11;
							VAR_ParameterWriter.fbClientDataExcha.nbExpectedChar := 6;
							
						36:	(*Film to run*)
							VAR_ParameterWriter.fbClientDataExcha.txBuffer[0]:=16#07;
							VAR_ParameterWriter.fbClientDataExcha.txBuffer[1]:=16#00;
							VAR_ParameterWriter.fbClientDataExcha.txBuffer[2]:= F_ToASC('U');
							VAR_ParameterWriter.fbClientDataExcha.txBuffer[3]:= F_ToASC('G');
							VAR_ParameterWriter.fbClientDataExcha.txBuffer[4]:= 16#00; (*n° de paramètre*)
							TEMP_DWORD := 16#01; (*film n°1*)
							MEMCPY(ADR(VAR_ParameterWriter.fbClientDataExcha.txBuffer[5]),ADR(TEMP_DWORD),4);
							VAR_ParameterWriter.fbClientDataExcha.txBuffer[9] := VAR_ParameterWriter.fbClientDataExcha.txBuffer[2] +
												VAR_ParameterWriter.fbClientDataExcha.txBuffer[3] +
												VAR_ParameterWriter.fbClientDataExcha.txBuffer[4] +
												VAR_ParameterWriter.fbClientDataExcha.txBuffer[5] +
												VAR_ParameterWriter.fbClientDataExcha.txBuffer[6] +
												VAR_ParameterWriter.fbClientDataExcha.txBuffer[7] +
												VAR_ParameterWriter.fbClientDataExcha.txBuffer[8];
							VAR_ParameterWriter.fbClientDataExcha.nbTransmittedChar := 10;
							VAR_ParameterWriter.fbClientDataExcha.nbExpectedChar := 6;
				END_CASE

			VAR_ParameterWriter.fbClientDataExcha(
								hSocket 		:= VAR_ParameterWriter.hSocket,
								bExecute 	:= TRUE,
								PRM_RECEIVE_POLLING_TIME:= T#1s, (*temporisation de polling de réception*)
								PRM_RECEIVE_TIMEOUT	:= T#10s);	(*temporisation de timeout de communication*)
			VAR_ParameterWriter.eStep := CLIENT_STATE_DATAEXCHA_WAIT;
		END_IF

	CLIENT_STATE_DATAEXCHA_WAIT:	(*Etape 4 - Attente de la fin de l'échange*)
		VAR_ParameterWriter.fbClientDataExcha( bExecute := FALSE );
		IF NOT VAR_ParameterWriter.fbClientDataExcha.bBusy THEN
			IF NOT VAR_ParameterWriter.fbClientDataExcha.bError THEN
				VAR_ParameterWriter.eStep 		:= CLIENT_STATE_DATA_ANALYSE;
			ELSE
				(* possible errors are logged inside of fbClientDataExcha function block *)
				VAR_ParameterWriter.nStepInError := 4;
				VAR_ParameterWriter.nErrId := 	VAR_ParameterWriter.fbClientDataExcha.nErrId;	(*n° d'erreur hérité de la fonction Fb_clientDataExchange*)
				VAR_ParameterWriter.ErrDescription :=	CONCAT(
												CONCAT(VAR_ParameterWriter.fbClientDataExcha.ErrDescription, ' '),
												CONCAT(' -Trame: ',UDINT_TO_STRING(VAR_ParameterWriter.nRequest))
												);
				VAR_ParameterWriter.eStep :=	CLIENT_STATE_ERROR;
			END_IF
		END_IF
	CLIENT_STATE_DATA_ANALYSE:	(*Etape 5 - Analyse des données reçues*)
		(*Contrôle que réponse ne comporte pas une erreur*)
		IF (VAR_ParameterWriter.fbClientDataExcha.rxBuffer[2] = 16#80) THEN
				VAR_ParameterWriter.nStepInError := 5;
				VAR_ParameterWriter.nErrId :=  1;
				VAR_ParameterWriter.ErrDescription := CONCAT(
								CONCAT( 'PACKET ERROR : ',F_ToCHR( VAR_ParameterWriter.fbClientDataExcha.RxBuffer[6])),
								CONCAT(' -Trame: ',UDINT_TO_STRING(VAR_ParameterWriter.nRequest))
								);
				VAR_ParameterWriter.eStep :=	CLIENT_STATE_ERROR;
		ELSE
			VAR_LOAD_PARAM := FALSE;										(*on refait tomber la commande*)
			VAR_ParameterWriter.nRequest := VAR_ParameterWriter.nRequest + 1;	(*incrémentation du n° de trame*)
			IF VAR_ParameterWriter.nRequest = 37 THEN
					VAR_ParameterWriter.nRequest := 0;
					STATE_Prog_Layer_OK := TRUE;
			END_IF
			VAR_ParameterWriter.eStep :=	CLIENT_STATE_IDLE;
		END_IF

	CLIENT_STATE_CLOSE_START:	(*Etape 6 - déclenchement fermeture du port*)
		VAR_ParameterWriter.fbClose( bExecute := FALSE );
		VAR_ParameterWriter.fbClose(
				hSocket:= VAR_ParameterWriter.hSocket,
				bExecute:= TRUE );
		VAR_ParameterWriter.eStep := CLIENT_STATE_CLOSE_WAIT;

	CLIENT_STATE_CLOSE_WAIT: (*Etape 7 - attente de la fermeture du port*)
		VAR_ParameterWriter.fbClose( bExecute := FALSE );
		IF NOT VAR_ParameterWriter.fbClose.bBusy THEN
			VAR_ParameterWriter.bConnected := FALSE;
			MEMSET( ADR(hSocket), 0, SIZEOF(hSocket));
			IF VAR_ParameterWriter.fbClose.bError THEN
				VAR_ParameterWriter.nErrId := VAR_ParameterWriter.fbClose.nErrId;
				VAR_ParameterWriter.nStepInError := 7;
				VAR_ParameterWriter.ErrDescription := CONCAT('FbClose Error : ', UDINT_TO_STRING(VAR_ParameterWriter.fbClose.nErrId));
				VAR_ParameterWriter.eStep := CLIENT_STATE_ERROR;
			ELSE
				VAR_ParameterWriter.bBusy := FALSE;
				VAR_ParameterWriter.bError := FALSE;
				VAR_ParameterWriter.nErrId := 0;
				VAR_ParameterWriter.eStep := CLIENT_STATE_IDLE;
			END_IF
		END_IF

	CLIENT_STATE_ERROR: (* Etape 8 : Error step *)
		VAR_ParameterWriter.bError := TRUE;
		IF VAR_ParameterWriter.bConnected THEN
			VAR_ParameterWriter.eStep := CLIENT_STATE_CLOSE_START;
		ELSE
			VAR_ParameterWriter.bBusy := FALSE;
			//IF DEF_COM_PARAMETER.AR_DEF THEN
				VAR_ParameterWriter.eStep := CLIENT_STATE_IDLE;
			//END_IF
		END_IF
END_CASE
END_ACTION

ACTION COM_STATUS:
CASE VAR_StatusReader.eStep OF
	CLIENT_STATE_IDLE:		(*Etape 0 - sequence d'échange à l'arrêt*)
		(*si autorisé ou exclusif si connecté*)
		IF VAR_StatusReader.bEnable XOR VAR_StatusReader.bConnected THEN
			VAR_StatusReader.bBusy := TRUE;
			VAR_StatusReader.bError := FALSE;
			VAR_StatusReader.nErrid := 0;
			IF VAR_StatusReader.bEnable THEN
				VAR_StatusReader.fbConnectTON( IN := FALSE );
				VAR_StatusReader.eStep := CLIENT_STATE_CONNECT_START;
			ELSE
				VAR_StatusReader.eStep := CLIENT_STATE_CLOSE_START;
			END_IF
		ELSIF VAR_StatusReader.bConnected THEN
			VAR_StatusReader.fbDataExchaTON( IN := FALSE );
			VAR_StatusReader.eStep := CLIENT_STATE_DATAEXCHA_START;
		ELSE
			VAR_StatusReader.bBusy := FALSE;
		END_IF

	CLIENT_STATE_CONNECT_START: (*Etape 1 - connexion au port*)
		(*temporisation de reconnexion*)
		VAR_StatusReader.fbConnectTON( IN := TRUE, PT := VAR_StatusReader.connectTime);
		(*si tempo de reconnexion ok*)
		IF VAR_StatusReader.fbConnectTON.Q THEN
			VAR_StatusReader.fbConnectTON( IN := FALSE );
			VAR_StatusReader.fbConnect(  bExecute := FALSE  );
			VAR_StatusReader.fbConnect(
						sRemoteHost		:= CONF_sRemoteHost,
						nRemotePort		:= CONF_nRemotePort,
						 sSrvNetId		:= '',
						bExecute		:= TRUE );
			VAR_StatusReader.eStep := CLIENT_STATE_CONNECT_WAIT;
			VAR_StatusReader.nRequest := 0; (*reinitalisation du n° de requete à 0*)
			VAR_StatusReader.Compteur_connection := VAR_StatusReader.Compteur_connection + 1;
		END_IF

	CLIENT_STATE_CONNECT_WAIT:	(*Etape 2 - attente connexion ok*)
		VAR_StatusReader.fbConnect( bExecute := FALSE );
		IF NOT VAR_StatusReader.fbConnect.bBusy THEN
			IF NOT VAR_StatusReader.fbConnect.bError THEN
				VAR_StatusReader.bConnected 	:= TRUE;
				VAR_StatusReader.hSocket 	:= VAR_StatusReader.fbConnect.hSocket;
				VAR_StatusReader.eStep 		:= CLIENT_STATE_IDLE;
				Def_connect_com_status := FALSE;
			ELSE
				(*LogError( 'FB_SocketConnect', fbConnect.nErrId );*)
				VAR_StatusReader.nErrId := VAR_StatusReader.fbConnect.nErrId;
				VAR_StatusReader.nStepInError  := 2;
				VAR_StatusReader.ErrDescription := CONCAT('FbConnect Error : ', UDINT_TO_STRING(VAR_StatusReader.fbConnect.nErrId));
				VAR_StatusReader.eStep := CLIENT_STATE_ERROR;
				Def_connect_com_status := TRUE;
			END_IF
		END_IF

	CLIENT_STATE_DATAEXCHA_START:	(*Etape 3 - lancement des échanges*)
		VAR_StatusReader.fbDataExchaTON( IN := TRUE, PT := VAR_StatusReader.ExchangeCycleTime );
		IF VAR_StatusReader.fbDataExchaTON.Q THEN
			VAR_StatusReader.fbDataExchaTON( IN := FALSE );
			VAR_StatusReader.fbClientDataExcha( bExecute := FALSE );

			CASE VAR_StatusReader.nRequest  OF
			0:
				(*Current Rate - S1*)
				VAR_StatusReader.fbClientDataExcha.txBuffer[0]:=16#02;
				VAR_StatusReader.fbClientDataExcha.txBuffer[1]:=16#00;
				VAR_StatusReader.fbClientDataExcha.txBuffer[2]:= F_ToASC('S');
				VAR_StatusReader.fbClientDataExcha.txBuffer[3]:= 16#01;
				VAR_StatusReader.fbClientDataExcha.txBuffer[4]:= VAR_StatusReader.fbClientDataExcha.txBuffer[2] +
															VAR_StatusReader.fbClientDataExcha.txBuffer[3];
				VAR_StatusReader.fbClientDataExcha.nbTransmittedChar := 5;
				VAR_StatusReader.fbClientDataExcha.nbExpectedChar := 10;
			1:
				(*Process Information - S0*)
				VAR_StatusReader.fbClientDataExcha.txBuffer[0]:=16#03;
				VAR_StatusReader.fbClientDataExcha.txBuffer[1]:=16#00;
				VAR_StatusReader.fbClientDataExcha.txBuffer[2]:= F_ToASC('S');
				VAR_StatusReader.fbClientDataExcha.txBuffer[3]:= 16#00;
				VAR_StatusReader.fbClientDataExcha.txBuffer[4]:= STATE_Timer_Tick;
				VAR_StatusReader.fbClientDataExcha.txBuffer[5]:= VAR_StatusReader.fbClientDataExcha.txBuffer[2] +
															VAR_StatusReader.fbClientDataExcha.txBuffer[3] +
															VAR_StatusReader.fbClientDataExcha.txBuffer[4];
				VAR_StatusReader.fbClientDataExcha.nbTransmittedChar := 6;
				VAR_StatusReader.fbClientDataExcha.nbExpectedChar := 30;

			2:	(*Crystal Life - S9*)
				VAR_StatusReader.fbClientDataExcha.txBuffer[0]:= 16#02;
				VAR_StatusReader.fbClientDataExcha.txBuffer[1]:=16#00;
				VAR_StatusReader.fbClientDataExcha.txBuffer[2]:= F_ToASC('S');
				VAR_StatusReader.fbClientDataExcha.txBuffer[3]:= 16#09;  (*09*)
				VAR_StatusReader.fbClientDataExcha.txBuffer[4]:= VAR_StatusReader.fbClientDataExcha.txBuffer[2] +
															VAR_StatusReader.fbClientDataExcha.txBuffer[3];
				VAR_StatusReader.fbClientDataExcha.nbTransmittedChar := 5;
				VAR_StatusReader.fbClientDataExcha.nbExpectedChar := 7;

			3:	(*Etat STOP*)
				VAR_StatusReader.fbClientDataExcha.txBuffer[0]:=16#02;
				VAR_StatusReader.fbClientDataExcha.txBuffer[1]:=16#00;
				VAR_StatusReader.fbClientDataExcha.txBuffer[2]:= F_ToASC('S');
				VAR_StatusReader.fbClientDataExcha.txBuffer[3]:=16#12;
				VAR_StatusReader.fbClientDataExcha.txBuffer[4]:= VAR_StatusReader.fbClientDataExcha.txBuffer[2] +
															VAR_StatusReader.fbClientDataExcha.txBuffer[3];
				VAR_StatusReader.fbClientDataExcha.nbTransmittedChar := 5;
				VAR_StatusReader.fbClientDataExcha.nbExpectedChar := 7;

			4: 	(*etat des entrées de l'XTC*)
				VAR_StatusReader.fbClientDataExcha.txBuffer[0]:=16#02;
				VAR_StatusReader.fbClientDataExcha.txBuffer[1]:=16#00;
				VAR_StatusReader.fbClientDataExcha.txBuffer[2]:= F_ToASC('S');
				VAR_StatusReader.fbClientDataExcha.txBuffer[3]:=16#0C;
				VAR_StatusReader.fbClientDataExcha.txBuffer[4]:= VAR_StatusReader.fbClientDataExcha.txBuffer[2] +
															VAR_StatusReader.fbClientDataExcha.txBuffer[3];
				VAR_StatusReader.fbClientDataExcha.nbTransmittedChar := 5;

			END_CASE

			VAR_StatusReader.fbClientDataExcha(
								hSocket 		:= VAR_StatusReader.hSocket,
								bExecute 	:= TRUE,
								PRM_RECEIVE_POLLING_TIME:= T#1s, (*temporisation de polling de réception*)
								PRM_RECEIVE_TIMEOUT	:= T#10s);	(*temporisation de timeout de communication*)
			VAR_StatusReader.eStep := CLIENT_STATE_DATAEXCHA_WAIT;
		END_IF

	CLIENT_STATE_DATAEXCHA_WAIT:	(*Etape 4 - Attente de la fin de l'échange*)
		VAR_StatusReader.fbClientDataExcha( bExecute := FALSE );
		IF NOT VAR_StatusReader.fbClientDataExcha.bBusy THEN
			IF NOT VAR_StatusReader.fbClientDataExcha.bError THEN
				VAR_StatusReader.eStep 		:= CLIENT_STATE_DATA_ANALYSE;
			ELSE
				(* possible errors are logged inside of fbClientDataExcha function block *)
				VAR_StatusReader.nStepInError := 4;
				VAR_StatusReader.nErrId := 	VAR_StatusReader.fbClientDataExcha.nErrId;	(*n° d'erreur hérité de la fonction Fb_clientDataExchange*)
				VAR_StatusReader.ErrDescription :=	CONCAT(
												CONCAT(VAR_StatusReader.fbClientDataExcha.ErrDescription, ' '),
												CONCAT(' -Trame: ',UDINT_TO_STRING(VAR_StatusReader.nRequest))
												);
				VAR_StatusReader.eStep :=	CLIENT_STATE_ERROR;
			END_IF
		END_IF
	CLIENT_STATE_DATA_ANALYSE:	(*Etape 5 - Analyse des données reçues*)
		(*si retour d'une trame signalant une erreur*)
		IF (VAR_StatusReader.fbClientDataExcha.rxBuffer[2] = 16#80) THEN
				VAR_StatusReader.nStepInError := 5;
				VAR_StatusReader.nErrId :=  1;
				VAR_StatusReader.ErrDescription := CONCAT(
								CONCAT( 'PACKET ERROR : ',F_ToCHR( VAR_StatusReader.fbClientDataExcha.RxBuffer[6])),
								CONCAT(' -Trame: ',UDINT_TO_STRING(VAR_StatusReader.nRequest))
								);
				VAR_StatusReader.eStep :=	CLIENT_STATE_ERROR;
		ELSE
			CASE VAR_StatusReader.nRequest  OF
				0:
					STATE_Timer_Tick:= VAR_StatusReader.fbClientDataExcha.RxBuffer[3];
					(*Récuperation de la vitesse d'évaporation*)
					MEMCPY(ADR(STATE_Rate),ADR(VAR_StatusReader.fbClientDataExcha.rxBuffer[5]),4);
				1:
					STATE_Timer_Tick:= VAR_StatusReader.fbClientDataExcha.rxBuffer[3];		(*Récuperation de la valeur du timer tick*)
					STATE_Sensor_Fail:= VAR_StatusReader.fbClientDataExcha.rxBuffer[5].0;		(*Etat du Quartz*)
					STATE_NPHASE := VAR_StatusReader.fbClientDataExcha.rxBuffer[6];		(*Phase en cours*)
					CASE	STATE_NPHASE OF
							0:
								STATE_Phase:= 'Ready';
							1:
								STATE_Phase:= 'Crucible Switch';
							2:
								STATE_Phase:= 'Rise 1';
							3:
								STATE_Phase:= 'Soak 1';
							4:
								STATE_Phase:= 'Rise 2';
							5:
								STATE_Phase:= 'Soak 2';
							6:
								STATE_Phase:= 'Shutter Delay';
							7:
								STATE_Phase:= 'Deposit';
							8:
								STATE_Phase:= 'Rate Ramp';
							9:
								STATE_Phase:= 'Manual';
							10:
								STATE_Phase:= 'Time Power';
							11:
								STATE_Phase:= 'Idle Ramp';
							12:
								STATE_Phase:= 'Idle';
				END_CASE
				STATE_Active_Sensor:= VAR_StatusReader.fbClientDataExcha.rxBuffer[7];
				STATE_Active_Crystal:= VAR_StatusReader.fbClientDataExcha.rxBuffer[8];
				(*Récuperation de la vitesse d'évaporation*)
				MEMCPY(ADR(STATE_Rate),ADR(VAR_StatusReader.fbClientDataExcha.rxBuffer[9]),4);
				(*Récuperation de l'épaisseur*)
				MEMCPY(ADR(STATE_Thickness),ADR(VAR_StatusReader.fbClientDataExcha.rxBuffer[13]),4);
				(*Récupération de la puissance*)
				MEMCPY(ADR(STATE_Power),ADR(VAR_StatusReader.fbClientDataExcha.rxBuffer[17]),4);
				(*Récuperation de la déviation de vitesse*)
				MEMCPY(ADR(STATE_Rate_Deviation),ADR(VAR_StatusReader.fbClientDataExcha.rxBuffer[21]),4);
				(*Récuperation de la fréquence*)
				MEMCPY(ADR(temp_dword),ADR(VAR_StatusReader.fbClientDataExcha.rxBuffer[25]),4);
				STATE_Frequency := temp_dword * VAR_Freq_Multiplieur;
			2:
				(*Récuperation de la durée de vie du Quartz*)
				STATE_Crystal_Life:= VAR_StatusReader.fbClientDataExcha.rxBuffer[5];
			3:
				STATE_STOP	:=	BYTE_TO_BOOL(VAR_StatusReader.fbClientDataExcha.rxBuffer[5]);

		END_CASE
		VAR_StatusReader.nRequest := VAR_StatusReader.nRequest + 1;	(*incrémentation du n° de trame*)
		IF VAR_StatusReader.nRequest = 4 THEN
			VAR_StatusReader.nRequest := 0;
		END_IF
		VAR_StatusReader.eStep :=	CLIENT_STATE_IDLE;
	END_IF

	CLIENT_STATE_CLOSE_START:	(*Etape 6 - déclenchement fermeture du port*)
		VAR_StatusReader.fbClose( bExecute := FALSE );
		VAR_StatusReader.fbClose(
				hSocket:= VAR_StatusReader.hSocket,
				bExecute:= TRUE );
		VAR_StatusReader.eStep := CLIENT_STATE_CLOSE_WAIT;

	CLIENT_STATE_CLOSE_WAIT: (*Etape 7 - attente de la fermeture du port*)
		VAR_StatusReader.fbClose( bExecute := FALSE );
		IF NOT VAR_StatusReader.fbClose.bBusy THEN
			VAR_StatusReader.bConnected := FALSE;
			MEMSET( ADR(hSocket), 0, SIZEOF(hSocket));
			IF VAR_StatusReader.fbClose.bError THEN
				VAR_StatusReader.nErrId := VAR_StatusReader.fbClose.nErrId;
				VAR_StatusReader.nStepInError := 7;
				VAR_StatusReader.ErrDescription := CONCAT('FbClose Error : ', UDINT_TO_STRING(VAR_StatusReader.fbClose.nErrId));
				VAR_StatusReader.eStep := CLIENT_STATE_ERROR;
			ELSE
				VAR_StatusReader.bBusy := FALSE;
				VAR_StatusReader.bError := FALSE;
				VAR_StatusReader.nErrId := 0;
				VAR_StatusReader.eStep := CLIENT_STATE_IDLE;
			END_IF
		END_IF

	CLIENT_STATE_ERROR: (* Etape 8 : Error step *)
		VAR_StatusReader.bError := TRUE;
		IF VAR_StatusReader.bConnected THEN
			VAR_StatusReader.eStep := CLIENT_STATE_CLOSE_START;
		ELSE
			VAR_StatusReader.bBusy := FALSE;
			//IF DEF_COM_STATUS.AR_DEF THEN
				VAR_StatusReader.eStep := CLIENT_STATE_IDLE;
			//END_IF
		END_IF
END_CASE
END_ACTION

ACTION POST:
(*Action G7 de gestion*)
(*étape 1 - Récupération des informations XTC*)
VAR_StatusReader.bEnable := OP_Gest.Etape.1;

(*étape 3 - Chargement des paramètres XTC*)
VAR_ParameterWriter.bEnable :=  OP_Gest.Etape.3;

(*étape 6 - Envoie d'une commande XTC*)
VAR_CommandWriter.bEnable := OP_Gest.Etape.6;


(*Défaut de Communication*)
IF (VAR_StatusReader.eStep = CLIENT_STATE_ERROR) AND NOT (VAR_StatusReader.nStepInError  = 2) THEN
	Condition_def_com_status := TRUE;
ELSIF Def_connect_com_status AND (VAR_StatusReader.nStepInError  = 2) THEN
	Condition_def_com_status := TRUE;
ELSE
	Condition_def_com_status := FALSE;
END_IF

DEF_COM_STATUS.CONDITION:= Condition_def_com_status AND NOT I_Inhibe_Def;
DEF_COM_STATUS.DELAY:= T#0s;
DEF_COM_STATUS.VAL1 := VAR_StatusReader.ErrDescription;
DEF_COM_STATUS();

(*Défaut de Communication*)
IF (VAR_ParameterWriter.eStep = CLIENT_STATE_ERROR) AND NOT (VAR_ParameterWriter.nStepInError  = 2) THEN
	Condition_def_com_parameters := TRUE;
ELSIF Def_connect_com_parameters AND (VAR_ParameterWriter.nStepInError  = 2) THEN
	Condition_def_com_parameters := TRUE;
ELSE
	Condition_def_com_parameters := FALSE;
END_IF

DEF_COM_PARAMETER.CONDITION:= Condition_def_com_parameters AND NOT I_Inhibe_Def;
DEF_COM_PARAMETER.DELAY:= T#0s;
DEF_COM_PARAMETER.VAL1 := VAR_ParameterWriter.ErrDescription;
DEF_COM_PARAMETER();

(*Défaut de Communication*)
IF (VAR_CommandWriter.eStep = CLIENT_STATE_ERROR) AND NOT (VAR_CommandWriter.nStepInError  = 2) THEN
	Condition_def_com_command := TRUE;
ELSIF Def_connect_com_command AND (VAR_CommandWriter.nStepInError  = 2) THEN
	Condition_def_com_command := TRUE;
ELSE
	Condition_def_com_command := FALSE;
END_IF

DEF_COM_COMMAND.CONDITION:= Condition_def_com_command AND NOT I_Inhibe_Def;
DEF_COM_COMMAND.DELAY:= T#0s;
DEF_COM_COMMAND.VAL1 := VAR_CommandWriter.ErrDescription;
DEF_COM_COMMAND();


(*Indicateur driver en fonctionnement*)
TIMER_STATE_READY.IN := (VAR_StatusReader.bConnected OR VAR_CommandWriter.bConnected OR VAR_ParameterWriter.bConnected) AND NOT STATE_NOK;
TIMER_STATE_READY.PT := T#10S;
TIMER_STATE_READY();

STATE_READY:= TIMER_STATE_READY.Q;

(*Indicateur contrôleur NON OK*)
STATE_NOK:= DEF_COM_PARAMETER.DEF OR DEF_COM_COMMAND.DEF OR DEF_COM_STATUS.DEF;

(*RAZ Indicateur de programmation couche ok*)
IF OP_Gest.Etape.1 THEN
	STATE_Prog_Layer_OK := FALSE;
END_IF

(*RAZ Indicateur d'action ok*)
IF OP_Gest.Etape.1 THEN
	STATE_ACTION_OK := FALSE;
	STATE_RAZ_THICK_OK := FALSE;
	STATE_START_OK:=FALSE;
	STATE_STOP_OK:=FALSE;
	STATE_RESET_OK:=FALSE;
	STATE_SWITCH_XTAL_OK:=FALSE;
END_IF

(*Affectation sorties*)
OUT_STOP_STATE		:=	IN_CD31T;
OUT_END_OF_PROCESS	:=	IN_CD32T;
OUT_CRYSTAL_FAIL		:=	IN_CD33T;
OUT_ALARMS			:=	IN_CD34T;
OUT_CACHE_SRCE		:=	IN_CD35T;
OUT_CACHE_QUARTZ	:=	IN_CD36T;
OUT_POWER_SP		:=	IN_CD31Q;
END_ACTION

ACTION PRL:
(*Défaut*)
DEF_COM_STATUS.IdXML := '16';
DEF_COM_STATUS.TagXML := 1;

DEF_COM_PARAMETER.IdXML := '16';
DEF_COM_PARAMETER.TagXML := 2;

DEF_COM_COMMAND.IdXML := '16';
DEF_COM_COMMAND.TagXML := 3;

VAR_Freq_Multiplieur	:= 0.0034924596;

(*Reception des bit d'ordre de maintenance*)
RCP_M_Start := M_Start;
RCP_M_Stop := M_Stop;
RCP_M_Reset := M_reset;
RCP_M_RAZ_Thick := M_RAZ_Thick;
RCP_M_Load_param := M_Load_param;
RCP_M_Switch_Crystal := M_Switch_Crystal;

(*Gestion de la sortie de mode manuel*)
(*les demandes d'action en mode manuel en attente sont resetées*)
FD_Manual(CLK:= Manual);

(*********Réception des ordres externes**********)
(*********demande de start ********)
FM_CO_Start(CLK:= CO_START);
IF	(*(NOT CO_START AND NOT MANUAL)
	OR *)FD_Manual.Q
	OR RESET THEN
	VAR_Start:= FALSE;
END_IF
IF 	((FM_CO_Start.Q AND NOT MANUAL)
	OR (RCP_M_Start AND MANUAL))
	AND NOT RESET  THEN
	VAR_Start:= TRUE;
END_IF


(**********demande de stop*********)
FM_CO_Stop(CLK:= CO_STOP);
IF	(NOT CO_STOP AND NOT MANUAL)
	OR FD_Manual.Q OR RESET THEN
	VAR_Stop:= FALSE;
END_IF
IF 	((FM_CO_Stop.Q AND NOT MANUAL)
	OR (RCP_M_Stop AND MANUAL))
	AND NOT RESET  THEN
	VAR_Stop:= TRUE;
END_IF

(*demande de RAZ épaisseur*)
FM_CO_Raz_Thick(CLK:= CO_RAZ_THICK);
IF	(NOT CO_RAZ_THICK AND NOT MANUAL)
	OR FD_Manual.Q OR RESET THEN
	VAR_Raz_Thick:= FALSE;
END_IF
IF 	((FM_CO_Raz_Thick.Q AND NOT MANUAL)
	OR (RCP_M_Raz_Thick AND MANUAL))
	AND NOT RESET  THEN
	VAR_Raz_Thick:= TRUE;
END_IF

(*demande de reset du contrôleur*)
FM_CO_RESET_Ctrl(CLK:= CO_RESET_Ctrl);
IF	(NOT CO_RESET_Ctrl AND NOT MANUAL)
	OR FD_Manual.Q OR RESET THEN
	VAR_Reset:= FALSE;
END_IF
IF 	((FM_CO_RESET_Ctrl.Q AND NOT MANUAL)
	OR (RCP_M_Reset  AND MANUAL))
	AND NOT RESET  THEN
	VAR_Reset:= TRUE;
END_IF

(*demande de programmation de la couche*)
FM_CO_Load_Param(CLK:= CO_Load_Param);
IF	(NOT CO_LOAD_PARAM AND NOT MANUAL)
	OR FD_Manual.Q OR RESET THEN
	VAR_LOAD_PARAM:= FALSE;
END_IF
IF 	((FM_CO_Load_Param.Q AND NOT MANUAL)
	OR (RCP_M_Load_Param  AND MANUAL))
	AND NOT RESET  THEN
	VAR_LOAD_PARAM:= TRUE;
END_IF

(*demande de switch du crystal*)
FM_CO_Switch_Crystal(CLK:= CO_Switch_Crystal);
IF	(NOT CO_Switch_Crystal AND NOT MANUAL)
	OR FD_Manual.Q
	OR RESET THEN
	VAR_SWITCH_CRYSTAL:= FALSE;
END_IF
IF 	((FM_CO_Switch_Crystal.Q AND NOT MANUAL)
	OR (RCP_M_Switch_Crystal AND MANUAL))
	AND NOT RESET  THEN
	VAR_SWITCH_CRYSTAL:= TRUE;
END_IF

(*RAZ des bit de d'ordre en mode manuel*)
IF RCP_M_Start AND M_Start THEN
	M_START:=FALSE;
END_IF
IF RCP_M_Stop AND M_Stop THEN
	M_STOP:=FALSE;
END_IF
IF RCP_M_Reset AND M_reset THEN
	M_RESET:=FALSE;
END_IF
IF RCP_M_RAZ_Thick AND M_RAZ_Thick THEN
	M_RAZ_Thick:=FALSE;
END_IF
IF RCP_M_Load_param AND M_Load_param THEN
	M_Load_param := FALSE;
END_IF
IF RCP_M_Switch_Crystal AND M_Switch_Crystal THEN
	M_Switch_Crystal:=FALSE;
END_IF
END_ACTION

END_FUNCTION_BLOCK

// ---- POUs/Fonction/FONCTION EVAPORATION/BLOCK_EVAP.TcPOU
FUNCTION_BLOCK BLOCK_EVAP

(* Gestion évaporation *)

(****************historique des versions*****************************)

(* Version 0-0 - SD - VERSION INITIALE CT200 n°7 - 8157 *)
(* Version 1-0 - GV - Ajout Gestion du balayage (Demande de marche & Arrêt balayage)
				+ Ajout demande de changement de creuset
				+ Ajout Timer temps couche pour visualisation
				+ Gestion Time Power *)
(* Version 2.0 - HG - Ajout CONF_No_Sweep
				- Suppression du délais défaut pmin et pmax pour configuration externe*)
(*Version 3-0 - GV -  Ajout gestion demande ouverture cache + Arrêt HT sur changement creuset + Ajout Défaut de refroidissement - affaire 9070 - 07/2015*)
(*Version 4-0 - HG - Ajout option dépôt à puissance fixe avec puissance segment 8 et temps max de dépôt
					Front montant pour start controleur*)
(*Version 4-1 - GV - Modification mémorisation mem_power pour Idle ramp pour éviter que la puissance passe à zéro*)
(*Version 4-2 - GV - Modification mémorisation mem_power pour Idle ramp -> Ajout (OUT_POWER <> 0) pour eviter que la puissance passe a zero*)
(*Versiob 5-0 - HG - Raccord avec block 3.3 des machines récentes
						Ajout CO_Modif
						Ajout I_Maintien_Source
						Modification reset RQ_Switch_crucible sur op_stop lorsqu'arrêt couche avant même le démarrage de la source
						Pas de défaut Pmin si PRM_Pmin = 0*)
(*************************************************************************)

VAR_INPUT
(*information générale*)
	RESET:								BOOL;
	MANUAL:								BOOL;
	I_EVAP_ON:							BOOL;			(*Demande d'évaporation par le bloc empilement aprés la phase de préfusion*)
	I_END_DEPOSITION:					BOOL;			(*Demande d'arrêt du dépôt*)
	I_DEF_QZ_CTRL_RATE:					BOOL;
	I_TIME_POWER:						BOOL;			(*Permet d'inhiber le défaut du quartz de contrôle de l'épaisseur si Option time power*)
	CO_FIN_ETAPE:						BOOL;	
	CO_MODIF:							BOOL;			(*Modification en ligne - Prise en compte nouvelles rampes de préfusion*)
	I_THICKNESS:						REAL;			(*épaisseur globale déposée*)
	I_SWITCH_XTAL_OK:					BOOL;			(*Indique que le positionnement de la tête multiquartz à été effectué*)
	I_OUV_CACHE_SOURCE:					BOOL;			(*Entrée de demande d'ouverture cache par le contrôleur de dépôt*)
	I_MAINTIEN_SOURCE:					BOOL;			(*Entrée de maintien de la source provenant du Block_Step_Empilement*)

(*opération*)
	OP_Marche:							BLOCK_OPERATION;	(*opération marche du bloc evap*)
	OP_Stop:							BLOCK_OPERATION;	(*opération arrêt du bloc*)

(*Défauts*)
	DEF_Pmax:							PRCDEF;		(*Défaut dépassement puissance max*)
	DEF_Pmin:							PRCDEF;		(*Défaut dépassement puissance min pendant les phases de dépôt/d'ajustement*)
	DEF_TEMPS_MAX:						PRCDEF;		(*Défaut temps d'enveloppe du dépôt*)
	DEF_QZ_CTRL_RATE:					PRCDEF;		(*Défaut du quartz de contrôle de l'épaisseur*)
	DEF_REF:							PRCDEF;		(*Défaut de refroidissement *)

(*Entrée diverses*)
	I_cache_ouvert:						BOOL;		(*Entrée Cache source ouvert*)
	I_cache_ferme:						BOOL;		(*Entree Cache source fermé*)
 	I_ref_source_ok:					BOOL;		(*Retour de refroidissement de la source ok*)
	I_ref_mesure_ok:					BOOL;		(*Retour de refroidissement de la mesure ok*)
	I_retour_pos_creuset_ok:			BOOL;		(*Retour de positionnement du creuset ok*)
	I_HT_ON:							BOOL;		(*Retour HT on*)
	I_HT_OFF:							BOOL;		(*Retour HT Off*)
	I_FIL_ON:							BOOL;		(*Retour FIL On*)
	I_FIL_OFF:							BOOL;		(*Retour Fil Off*)
	I_SWEEP_ON:							BOOL;		(*Retour balayage en marche*)
	I_Power:							REAL;		(*puissance demandée par le controleur de dépôt pendant la phase d'évaporation en %*)
END_VAR


VAR_OUTPUT
	STATE_Segment:					USINT;			(*N° du segment en cours*)
	STATE_Temps_segment:			TIME;			(*Temps restant pour le segment en cours*)
	STATE_Temps_Phase:				TIME;			(*Temps restant pour la phase en cours : préparation / dépôt / cloture*)
	STATE_TEMPS_PREPARATION:		INT;			(*Temps de préparation total en seconde*)
	STATE_TEMPS_CLOTURE:			INT;			(*Temps de cloture total en seconde*)
	STATE_TEMPS_DEPOT:				INT;			(*Temps de dépôt estimé en fonction de la vitesse et de l'épaisseur attendue*)
	STATE_TEMPS_RESTANT_PREP:		INT;			(*Temps de préparation restant en seconde*)
	STATE_TEMPS_RESTANT_CLOT:		INT;			(*Temps de cloture restant en seconde*)
	STATE_TEMPS_RESTANT_DEPOT:		INT;			(*Temps restant de dépôt en seconde*)

	OUT_Power:							REAL;		(*Puissance demandée en %*)
	OUT_Cons_Pos_Qz:					INT;		(*Quartz à utiliser*)
	OUT_Start_Controleur:				BOOL;		(*Demande de start du controleur*)
	RQ_ouv_cache_IAD:					BOOL;		(*bit utilisé pour ouverture synchronisé du cache IAD*)
	RQ_Ref_source:						BOOL;		(*Demande de refroidissement de la source*)
	RQ_Ref_mesure:						BOOL;		(*Demande de refroidissement de la mesure*)
	RQ_Ouv_Cache_source:				BOOL;		(*Demande d'ouverture du cache*)
	RQ_marche_HT:						BOOL;		(*Demande de marche de la haute tension*)
	RQ_marche_FIL:						BOOL;		(*Demande de marche de la source à effet joule ou de la haute-tension*)
	RQ_marche_SWEEP:					BOOL;		(*Demande de marche du balayage*)
	RQ_Switch_Crucible:					BOOL;		(*Demande de changement de creuset*)
	RQ_Switch_Crystal:					BOOL;		(*Demande de switch tête multiquartz*)


	STATE_PREP_OK:					BOOL;		(*Phase de préparation ok*)
	STATE_EVAP:						BOOL;		(*Phase d'évaporation en cource*)
	STATE_CLOT_OK:					BOOL;
	STATE_AR:						BOOL;		(*Evaporation à l'arrêt*)
	STATE_PREFU:					BOOL;		(*Phase de préfusion en cours*)
	STATE_IDLE:						BOOL;		(*Phase de descente en cours*)
	STATE_END_DEPOT_PFIXE:			BOOL;		(*Fin dépot détecté sur puissance fixe, pour STEP_EMPILEMENT*)

END_VAR
VAR_INPUT PERSISTENT
(*Entité*)
	IsAssembly:							BOOL;		(*entité : fonction*)
	IdXML:								STRING;		(*nom entité : identifiant pour recherche dans dico*)
	TagXML:								UINT;		(*nom entité : identifiant pour recherche dans dico*)
	IdParent:							STRING;		(*MNEMO de l'appelant*)
	MNEMO:								STRING;		(*MNEMO de l'entité*)


(*Paramètres de configurations*)
	PRM_Thickness:						REAL;			(*Consigne d'épaisseur en kA°*)
	PRM_Rate:							REAL;			(*Consigne de vitesse de dépôt en A°/s*)
	PRM_PFixe:							BOOL;			(*Option dépôt à puissance fixe*)
	PRM_TPS_Max_PFixe:					UINT;			(*Temps max de dépôt si option puissance fixe*)
	PRM_TPS_SEGMENT:				ARRAY[0..10] OF INT;	(*Temps pour chaque segment*)
	PRM_PWR_SEGMENT:				ARRAY[0..10] OF REAL;	(*Puissance pour chaque segment*)
	PRM_GAIN:							REAL;			(*Parametre de gain*)
	PRM_INTEGRAL:						REAL;			(*Paramètre intégrale source*)
	PRM_DERIVEE:						REAL;			(*Paramètre derivée*)
	PRM_AUTO_SOAK2:						BOOL;			(*Option de calcul automatique de la valeur du segment 7*)
	PRM_PHASE_PREFFUSION:				USINT:=1;		(*N° de phase de préfusion, permet de savoir par quelle phase commencer, = à 1 par défaut*)
	PRM_PMAX:							REAL:= 10;		(*Puissance max pour la source*)
	PRM_PMIN:							REAL;			(*Puissance min pour la source*)
	PRM_TIMEPOWER:						BOOL;			(*Paramètre time power*)
	PRM_RETARD_FERM_CACHE:				REAL;			(*Paramètre de retard fermeture cache en s*)
	PRM_REOUV_CACHE:					REAL;			(*Temps pour réouverture du cache*)
	PRM_NCR:							USINT;			(*N° de creuset selectionné*)
	PRM_NBAL:							USINT;			(*N° de programme de balayage*)
	PRM_HT:								REAL;			(*consigne HT*)

	PRM_CRYSTAL_POSITION:				INT;		(*Numéro du crystal à utiliser pour la tête MultiQuartz, 1 à 6 *)

	PRM_Transfer_Tooling:				REAL;		(*Facteur de correction du Quartz d'ajustement de la vitesse en fin de phase de préfusion*)

	PRM_MULTIPOINT:						BOOL;		(*Indique s'il y a utilisation de plusieurs Quartz pour le contrôle vitesse, donnée par l'éditeur*)
	PRM_MULTI_QUARTZ:					BOOL;		(*Indique s'il y a une tête multiquartz*)

	PRM_NQz_Rate:						USINT;					(*N° de quartz qui controle la vitesse de dépot de la source en mode MonoPoint*)
	PRM_NQz_MultiPoint:					ARRAY[0..7] OF USINT;		(*N° des Quartz utilisés pour contrôle de la vitesse de dépôt en mode MultiPoint*)
	PRM_Num_Transfer_Sensor:			BYTE;					(*Numéro du capteur utilisé pour le Quartz de contrôle pendant phase de préfusion*)

	PRM_SOAK2_POWER:					REAL;		(*Puissance soak power 2 à transmettre au controleur de dépôt*)
	PRM_Quartz_Cache_Source:			BOOL;		(*Indique s'il y a un Quartz de contrôle sous le cache source*)
	PRM_SHUTTER_Option:					BOOL;		(*Option d'utilisation du Quartz de transfert, Quartz sous le cache source*)
	PRM_CTRL_DELAY_TIME:				INT;		(*Délai en secondes entre l'ouverture du cache source et prise de contrôle de la vitesse d'évaporation*)
(*	PRM_CTRL_DELAY:						BOOL;		(*Option d'utilisation du Quartz de transfert, Quartz sous le cache source*)*)

(*Parametres quartz*)
	PRM_Quality_Percent:					USINT;		(*Déviation max de la fréquence*)
	PRM_Quality_Counts:						USINT;		(*Nombre de déviation de la fréquence autorisée*)
	PRM_Stability_Single:					UINT;		(*Déviation de la fréquence*)
	PRM_Stability_Total:					UINT;		(*Déviation total de la fréquence*)

	PRM_Shutter_Delay_Acc:					USINT;

(*Parametres pour la nouvelle vitesse*)
	PRM_New_Rate:						REAL;		(*Nouvelle consigne de vitesse en A°/s*)
	PRM_Rate_Ramp_Time:					UINT;		(*Temps de monté à la nouvelle consigne de vitesse en secondes*)
	PRM_Thick_SP:						REAL;		(*Epaisseur qui déclenche la nouvelle vitesse en kA°*)


(*configuration Surveillance du dépôt*)
	PRM_TPS_MIN_SURV_DEPOT:			INT;		(*Temps mini pour la surveillance du temps de depot*)
(*	PRM_SEUIL_TEMPS_DEPOT:			REAL;		(*Seuil temps de dépôt théorique à partir duquel on applique un facteur au temps de dépôt théorique*)*)
	PRM_FACTEUR_TEMPS_DEPOT:		REAL;		(*Facteur du temps théorique*)

(*Paramètres de configuration matériel*)
	CONF_No_Sweep:					BOOL;
END_VAR

VAR_TEMP
	FLAG_PMAX:						BOOL;		(*Flag puissance max atteinte*)
	FLAG_PMIN:						BOOL;		(*Flag puissance min atteinte*)
END_VAR

VAR_IN_OUT
	CONS_NCR:						USINT;		(*Consigne n° de creuset à utiliser*)
	CONS_NBAL:						USINT;		(*Consigne n° de programme de balayage*)
	CONS_HT:						REAL;
END_VAR

VAR
	MEM_POWER:							REAL;		(*Variable mémoire puissance*)
	TIMER_SEGMENT:						ARRAY[0..10] OF TON;
	I:									USINT;
	VAR_Pi:								REAL;		(*utilisé pour calcul*)
	VAR_Pf:								REAL;		(*utilisé pour calcul*)
	VAR_Time:							REAL;		(*Utilisé pour calcul*)
	VAR_Tseg:							REAL;		(*Utilisé pour calcul*)
	VAR_Mem_Creuset:					USINT;		(*Variable mémoire du n° de creuset utilisé lors de la dernière couche*)
	TIMER_RETARD_FCACHE:			TP;
	TIMER_RETARD_OCACHE:			TON;
	FM_ETAPE3_MARCHE:				R_TRIG;
	FM_ETAPE14_MARCHE:				R_TRIG;
	VAR_RETARD_FERM_CACHE:			BOOL;
	TIMER_Prise_Controle:			TON;
	TIMER_Temps_Couche:				TON;
	TIMER_Start_Controleur:			TP;
	FM_CO_Modif:					R_TRIG;
END_VAR

PRL();

ACT_MARCHE();
ACT_STOP();

POST();

ACTION ACT_MARCHE:
(* OPERATION marche évaporation*)

OP_MARCHE(
	ON_AUTO_INT:= ,
	CTRL_PLC:= TRUE,
	RESET:= RESET ,
	MANUAL:= MANUAL,
	ENABLE_INT:= TRUE,
	RESTART_ENABLE_IF_OK:=TRUE ,
	N_STEP_OP_OK:= 16,
	N_STEP_OP_NOK:=0 );


OP_MARCHE.PRL();

(*GRAFCET*)
(* initialisation du grafcet*)
IF 		OP_Marche.ETAPE = 0 THEN
				OP_Marche.ETAPE.0 := TRUE;
(*repositionnement sur étape 0*)
ELSIF	MANUAL OR RESET OR OP_Stop.Etape.1	THEN
				OP_Marche.ETAPE := 0;			(*RAZ grafcet*)
				OP_Marche.ETAPE.0:=TRUE;
(*étape 0-1*)
ELSIF 	OP_Marche.ETAPE.0
		AND OP_Marche.MARCHE_OP   THEN
				OP_Marche.ETAPE.1:=TRUE;
				OP_Marche.ETAPE.0:=FALSE;
(*étape 5.6.7.8.9.10.11.12.13 - 14 fin de couche*)
ELSIF	(OP_Marche.ETAPE.5 OR
		OP_Marche.ETAPE.6 OR
		OP_Marche.ETAPE.7 OR
		OP_Marche.ETAPE.8 OR
		OP_Marche.ETAPE.9 OR
		OP_Marche.Etape.10 OR
		OP_Marche.Etape.11 OR
		OP_Marche.Etape.12 OR
		OP_Marche.Etape.13 )
		AND CO_FIN_ETAPE THEN
				OP_Marche.Etape.14:=TRUE;
				OP_Marche.Etape.5:=FALSE;
				OP_Marche.Etape.6:=FALSE;
				OP_Marche.Etape.7:=FALSE;
				OP_Marche.Etape.8:=FALSE;
				OP_Marche.Etape.9:=FALSE;
				OP_Marche.Etape.10:=FALSE;
				OP_Marche.Etape.11:=FALSE;
				OP_Marche.Etape.12:=FALSE;
				OP_Marche.Etape.13:=FALSE;
(*étape 1.2.3.4. - 16 - fin de couche*)
ELSIF	(OP_Marche.ETAPE.1 OR
		OP_Marche.ETAPE.2 OR
		OP_Marche.ETAPE.3 OR
		OP_Marche.ETAPE.4 )
		AND CO_FIN_ETAPE THEN
				OP_Marche.Etape.16:=TRUE;
				OP_Marche.Etape.1:=FALSE;
				OP_Marche.Etape.2:=FALSE;
				OP_Marche.Etape.3:=FALSE;
				OP_Marche.Etape.4:=FALSE;

(*étape 1-2*)
ELSIF	OP_Marche.ETAPE.1
		AND OP_Stop.AR AND ((NOT (PRM_NCR = VAR_Mem_Creuset) AND I_HT_OFF AND I_FIL_OFF) OR (PRM_NCR = VAR_Mem_Creuset)) THEN
				OP_Marche.Etape.2:=TRUE;
				OP_Marche.Etape.1:=FALSE;
(*étape 2-17*)
ELSIF 	OP_Marche.Etape.2
		AND I_retour_pos_creuset_ok
		AND I_ref_mesure_ok
		AND I_ref_source_ok
		AND (I_SWITCH_XTAL_OK OR NOT PRM_MULTI_QUARTZ)
		 THEN
				OP_Marche.Etape.17:=TRUE;
				OP_Marche.Etape.2:=FALSE;
(*étape 17-3*)
ELSIF	OP_Marche.Etape.17
		AND (I_SWEEP_ON OR CONF_No_Sweep) THEN
				OP_Marche.Etape.3:=TRUE;
				OP_Marche.Etape.17:= FALSE;
(*étape 3-4*)
ELSIF	OP_Marche.ETAPE.3
		AND I_HT_ON THEN
				OP_Marche.Etape.4:=TRUE;
				OP_Marche.Etape.3:=FALSE;
(*étape 4-5*)
(*	La puissance n'a pas été maintenue et la phase de préfusion 0 est demandée- execution de la premiere rampe
	et du premier palier*)
ELSIF	OP_MARCHE.ETAPE.4 AND
		I_FIL_ON AND ( PRM_PHASE_PREFFUSION =1) AND NOT I_MAINTIEN_SOURCE THEN
				MEM_POWER := OUT_POWER;
				OP_Marche.Etape.5:=TRUE;
				OP_Marche.Etape.4:=FALSE;
(*étape 4-10*)
(*	La puissance a été maintenue ou la phase de préfusion 2 est demandée - passage au segment n°6*)
ELSIF	OP_MARCHE.ETAPE.4
		AND ( PRM_PHASE_PREFFUSION = 3) AND I_FIL_ON AND NOT I_MAINTIEN_SOURCE THEN
				MEM_POWER := OUT_POWER;
				OP_Marche.Etape.10:=TRUE;
				OP_Marche.Etape.4:=FALSE;
(*Etape 4-8*)
ELSIF	OP_MARCHE.ETAPE.4
		AND ( PRM_PHASE_PREFFUSION = 2) AND I_FIL_ON AND NOT I_MAINTIEN_SOURCE THEN
				MEM_POWER := OUT_POWER;
				OP_Marche.Etape.8:=TRUE;
				OP_Marche.Etape.4:=FALSE;		

(*Etape 4-6*)		
ELSIF	OP_MARCHE.ETAPE.4
		AND I_MAINTIEN_SOURCE AND I_FIL_ON THEN
				MEM_POWER := OUT_POWER;
				OP_Marche.Etape.6:=TRUE;
				OP_Marche.Etape.4:=FALSE;				
(*étape 5-6*)
ELSIF	OP_MARCHE.ETAPE.5
		AND TIMER_SEGMENT[1].Q THEN 			(*fin segment 1*)
				MEM_POWER := OUT_POWER;
				OP_MARCHE.Etape.6:=TRUE;
				OP_MARCHE.Etape.5:=FALSE;
(*étape 6-7*)
ELSIF	OP_MARCHE.ETAPE.6
		AND TIMER_SEGMENT[2].Q THEN 			(*fin segment 2*)
				MEM_POWER := OUT_POWER;
				OP_MARCHE.Etape.7:=TRUE;
				OP_MARCHE.Etape.6:=FALSE;
(*étape 7-8*)
ELSIF	OP_MARCHE.ETAPE.7
		AND TIMER_SEGMENT[3].Q THEN			(*fin segment 3*)
				MEM_POWER := OUT_POWER;
				OP_MARCHE.Etape.8:=TRUE;
				OP_MARCHE.Etape.7:=FALSE;
(*étape 8-9*)
ELSIF	OP_MARCHE.ETAPE.8
		AND TIMER_SEGMENT[4].Q THEN			(*fin segment 4*)
				MEM_POWER := OUT_POWER;
				OP_MARCHE.Etape.9:=TRUE;
				OP_MARCHE.Etape.8:=FALSE;
(*étape 9-10*)
ELSIF	OP_MARCHE.ETAPE.9
		AND TIMER_SEGMENT[5].Q THEN			(*fin segment 5*)
				MEM_POWER := OUT_POWER;
				OP_MARCHE.Etape.10:=TRUE;
				OP_MARCHE.Etape.9:=FALSE;
(*étape 10-11*)
ELSIF	OP_MARCHE.ETAPE.10
		AND TIMER_SEGMENT[6].Q THEN			(*fin segment 6*)
				MEM_POWER := OUT_POWER;
				OP_MARCHE.Etape.11:=TRUE;
				OP_MARCHE.Etape.10:=FALSE;
(*étape 11-12*)
ELSIF	OP_MARCHE.ETAPE.11
		AND TIMER_SEGMENT[7].Q THEN			(*fin segment 7*)
				MEM_POWER := OUT_POWER;
				OP_MARCHE.Etape.12:=TRUE;
				OP_MARCHE.Etape.11:=FALSE;

(*étape 12-13*)
ELSIF	OP_MARCHE.ETAPE.12
		AND I_EVAP_ON THEN						(*Demande START dépot par bloc empilement*)
				OP_MARCHE.Etape.13:=TRUE;
				OP_MARCHE.Etape.12:=FALSE;

(*Début du dépôt*)
(*étape 13-14*)
ELSIF	OP_MARCHE.ETAPE.13
		AND I_END_DEPOSITION THEN
				VAR_RETARD_FERM_CACHE:=TRUE;
				OP_MARCHE.Etape.14:=TRUE;
				OP_MARCHE.Etape.13:=FALSE;
(*étape 14-15*)
ELSIF	OP_MARCHE.ETAPE.14
		AND TIMER_SEGMENT[9].Q THEN
				MEM_POWER := OUT_POWER;
				OP_MARCHE.Etape.15:=TRUE;				(*Rampe de descente 1*)
				OP_MARCHE.Etape.14:=FALSE;
(*étape 15-16*)
ELSIF	OP_MARCHE.ETAPE.15
		AND TIMER_SEGMENT[10].Q THEN
				MEM_POWER := OUT_POWER;
				OP_MARCHE.Etape.16:=TRUE;				(*Rampe de descente 2*)
				OP_MARCHE.Etape.15:=FALSE;
(*étape 16-1*)
ELSIF	OP_MARCHE.ETAPE.16
		AND OP_MARCHE.MARCHE_OP  THEN
				MEM_POWER := OUT_POWER;
				OP_MARCHE.Etape.1:=TRUE;
				OP_MARCHE.Etape.16:=FALSE;

END_IF;

(*cloture du traitement de l'opération*)
OP_Marche.POST();
END_ACTION

ACTION ACT_STOP:
(* OPERATION d'arret d'évaporation*)
(* arrêt de l'opération*)

(*initialisation de l'opération*)
OP_STOP(
	ON_AUTO_INT:= ,
	CTRL_PLC:= TRUE,
	RESET:= RESET ,
	MANUAL:= MANUAL,
	ENABLE_INT:= TRUE,
	RESTART_ENABLE_IF_OK:=FALSE ,
	N_STEP_OP_OK:= 5,
	N_STEP_OP_NOK:=0 );


(*appel de l'action de préparation de l'opération*)
OP_STOP.PRL();

(*GRAFCET*)
(* initialisation du grafcet*)
IF 		OP_Stop.ETAPE = 0 THEN
				OP_Stop.ETAPE.0 := TRUE;
(*repositionnement sur étape 0*)
ELSIF	MANUAL OR Reset OR OP_Marche.Etape.1 THEN
				OP_Stop.ETAPE := 0;			(*RAZ grafcet*)
				OP_Stop.ETAPE.0:=TRUE;
(*étape 0-1*)
ELSIF 	OP_Stop.ETAPE.0
		AND OP_Stop.marche_op THEN
				OP_Stop.ETAPE.1:=TRUE;
				OP_Stop.ETAPE.0:=FALSE;
(*étape 1-2*)
ELSIF	OP_Stop.ETAPE.1
		AND OP_Marche.AR  THEN
				OP_Stop.Etape.2:=TRUE;
				OP_Stop.Etape.1:=FALSE;
(*étape 2-3*)
ELSIF 	OP_Stop.Etape.2
		AND I_FIL_OFF
		 THEN
				OP_Stop.Etape.3:=TRUE;
				OP_Stop.Etape.2:=FALSE;
(*étape 3-4*)
ELSIF 	OP_Stop.Etape.3
		AND I_HT_OFF
		 THEN
				OP_Stop.Etape.4:=TRUE;
				OP_Stop.Etape.3:=FALSE;
(*étape 4-5*)
ELSIF	OP_Stop.Etape.4
		(*AND (NOT I_SWEEP_ON OR CONF_No_Sweep)*)		(*Pas de commande d'arrêt du sweep*)
		THEN
				OP_Stop.Etape.5:=TRUE;
				OP_Stop.Etape.4:=FALSE;
END_IF;


(*cloture du traitement de l'opération*)
OP_Stop.POST();
END_ACTION

ACTION POST:
(*Gestion demandes*)
FM_CO_Modif(clk:=CO_modif);

(*************************************************)
(* GESTION PUISSANCE DE SORTIE     *)
(************************************************)
(*
FM_ETAPE14_MARCHE(CLK:=OP_marche.Etape.14);
IF FM_ETAPE14_MARCHE.Q THEN
	MEM_POWER := OUT_POWER;
END_IF
*)

IF OP_MARCHE.Etape.13 AND NOT I_END_DEPOSITION AND (OUT_POWER <> 0) THEN 
	MEM_POWER := OUT_POWER;
END_IF

(*initialisation des temporisations de segment*)
IF OP_MARCHE.Etape.1 OR FM_CO_Modif.Q THEN
		TIMER_SEGMENT[1].PT := INT_TO_TIME(PRM_TPS_SEGMENT[1])*1000;
		TIMER_SEGMENT[2].PT := INT_TO_TIME(PRM_TPS_SEGMENT[2])*1000;
		TIMER_SEGMENT[3].PT := INT_TO_TIME(PRM_TPS_SEGMENT[3])*1000;
		TIMER_SEGMENT[4].PT := INT_TO_TIME(PRM_TPS_SEGMENT[4])*1000;
		TIMER_SEGMENT[5].PT := INT_TO_TIME(PRM_TPS_SEGMENT[5])*1000;
		TIMER_SEGMENT[6].PT := INT_TO_TIME(PRM_TPS_SEGMENT[6])*1000;
		TIMER_SEGMENT[7].PT := INT_TO_TIME(PRM_TPS_SEGMENT[7])*1000;
		TIMER_SEGMENT[8].PT := INT_TO_TIME(PRM_TPS_SEGMENT[8])*1000;	(*Dépôt*)
		TIMER_SEGMENT[9].PT := INT_TO_TIME(PRM_TPS_SEGMENT[9])*1000;
		TIMER_SEGMENT[10].PT := INT_TO_TIME(PRM_TPS_SEGMENT[10])*1000;
END_IF

TIMER_SEGMENT[1].IN := OP_MARCHE.Etape.5;
TIMER_SEGMENT[2].IN := OP_MARCHE.Etape.6;
TIMER_SEGMENT[3].IN := OP_MARCHE.Etape.7;
TIMER_SEGMENT[4].IN := OP_MARCHE.Etape.8;
TIMER_SEGMENT[5].IN := OP_MARCHE.Etape.9;
TIMER_SEGMENT[6].IN := OP_MARCHE.Etape.10;
TIMER_SEGMENT[7].IN := OP_MARCHE.Etape.11;
TIMER_SEGMENT[8].IN := OP_MARCHE.Etape.13;
TIMER_SEGMENT[9].IN := OP_MARCHE.Etape.14;
TIMER_SEGMENT[10].IN := OP_MARCHE.Etape.15;

TIMER_SEGMENT[1]();
TIMER_SEGMENT[2]();
TIMER_SEGMENT[3]();
TIMER_SEGMENT[4]();
TIMER_SEGMENT[5]();
TIMER_SEGMENT[6]();
TIMER_SEGMENT[7]();
TIMER_SEGMENT[8]();
TIMER_SEGMENT[9]();
TIMER_SEGMENT[10]();

TIMER_Prise_Controle.IN := OP_MARCHE.Etape.13;
TIMER_Prise_Controle.PT :=T#3s;
TIMER_Prise_Controle();

(*Timer pour pour visualisation temps de la couche*)
TIMER_Temps_Couche (	PT:= T#30000m,
						IN := OP_MARCHE.Etape.13,);

(*Puissance appliquée en fin de préfusion*)
PRM_SOAK2_POWER:= PRM_PWR_SEGMENT[7];
(*Demande de switch crystal*)
RQ_Switch_Crystal:= OP_Marche.Etape.2 AND PRM_MULTI_QUARTZ;
(*Position à utiliser pour la tête multiquartz*)
OUT_Cons_Pos_Qz:= PRM_CRYSTAL_POSITION;

(*Calcul du temps total de préparation du dépôt*)
IF OP_Marche.Etape.1 OR FM_CO_Modif.Q THEN
(*	STATE_TEMPS_PREPARATION := 	PRM_TPS_SEGMENT[1] + PRM_TPS_SEGMENT[2] + PRM_TPS_SEGMENT[3] +
										PRM_TPS_SEGMENT[4] + PRM_TPS_SEGMENT[5] + PRM_TPS_SEGMENT[6] +
										PRM_TPS_SEGMENT[7];
*)
	IF PRM_PHASE_PREFFUSION  = 1 THEN
		STATE_TEMPS_PREPARATION := 		PRM_TPS_SEGMENT[1] + PRM_TPS_SEGMENT[2] + PRM_TPS_SEGMENT[3] +
										PRM_TPS_SEGMENT[4] + PRM_TPS_SEGMENT[5] + PRM_TPS_SEGMENT[6] +
										PRM_TPS_SEGMENT[7];
	END_IF
	IF PRM_PHASE_PREFFUSION = 2THEN
		STATE_TEMPS_PREPARATION := 		PRM_TPS_SEGMENT[4] + PRM_TPS_SEGMENT[5] + PRM_TPS_SEGMENT[6] +
										PRM_TPS_SEGMENT[7];
	END_IF
	IF PRM_PHASE_PREFFUSION = 3 THEN
		STATE_TEMPS_PREPARATION := 		PRM_TPS_SEGMENT[6] +
										PRM_TPS_SEGMENT[7];
	END_IF

	STATE_TEMPS_CLOTURE  :=	PRM_TPS_SEGMENT[9] + PRM_TPS_SEGMENT[10];		(*Temps de clôture estimé*)

	IF PRM_RATE > 0 THEN	(*On évite la division par 0*)
		IF PRM_New_Rate > 0 THEN	(*Calcul du temps théorique si nouvelle vitesse*)
			STATE_TEMPS_DEPOT	:=	REAL_TO_INT(((PRM_THICK_SP*1000) / PRM_Rate) + (((PRM_Thickness-PRM_Thick_SP)*1000) / PRM_New_Rate));
		ELSE
			STATE_TEMPS_DEPOT	:=	REAL_TO_INT((PRM_Thickness*1000) / PRM_Rate);		(*Temps de dépôt estimé, théorique*)
		END_IF
	END_IF

	STATE_TEMPS_RESTANT_CLOT 		:=	STATE_TEMPS_CLOTURE;
	STATE_TEMPS_RESTANT_PREP		:=	STATE_TEMPS_PREPARATION;
	STATE_TEMPS_RESTANT_DEPOT 	:=	STATE_TEMPS_DEPOT;
END_IF


(*ATTENTION Modif amory pour anticipation, il faut mettre à jour les temps lors de cloture pour pouvoir relancer l'évap*)
IF OP_Marche.Etape.16 OR OP_Marche.Etape.15 OR OP_Marche.Etape.14 OR OP_Marche.Etape.0 THEN
	IF PRM_PHASE_PREFFUSION  = 1 THEN
		STATE_TEMPS_PREPARATION := 		PRM_TPS_SEGMENT[1] + PRM_TPS_SEGMENT[2] + PRM_TPS_SEGMENT[3] +
										PRM_TPS_SEGMENT[4] + PRM_TPS_SEGMENT[5] + PRM_TPS_SEGMENT[6] +
										PRM_TPS_SEGMENT[7];
	END_IF
	IF PRM_PHASE_PREFFUSION = 2 THEN
		STATE_TEMPS_PREPARATION := 		PRM_TPS_SEGMENT[4] + PRM_TPS_SEGMENT[5] + PRM_TPS_SEGMENT[6] +
										PRM_TPS_SEGMENT[7];
	END_IF
	IF PRM_PHASE_PREFFUSION = 3 THEN
		STATE_TEMPS_PREPARATION := 		PRM_TPS_SEGMENT[6] +
										PRM_TPS_SEGMENT[7];
	END_IF
END_IF


(*Calcul de la consigne de puissance en % en fonction du segment en cours*)
CASE OP_MARCHE.STATUS OF
	5:
		STATE_Segment 	:= 	1;
		STATE_TEMPS_SEGMENT := TIMER_SEGMENT[1].PT - TIMER_SEGMENT[1].ET;

		CASE PRM_PHASE_PREFFUSION OF
			1:
				STATE_TEMPS_RESTANT_PREP := 	STATE_TEMPS_PREPARATION -
													TIME_TO_INT(TIMER_SEGMENT[1].ET / 1000);

			2,3:
				STATE_TEMPS_RESTANT_PREP :=	STATE_TEMPS_RESTANT_PREP;
		END_CASE

		STATE_TEMPS_RESTANT_CLOT := 	STATE_TEMPS_CLOTURE;
		STATE_Temps_Phase 		       := 	INT_TO_TIME(STATE_TEMPS_RESTANT_PREP) * 1000;

	6:
		STATE_Segment	:= 	2;
		STATE_TEMPS_SEGMENT := TIMER_SEGMENT[2].PT - TIMER_SEGMENT[2].ET;

		CASE PRM_PHASE_PREFFUSION OF
			1:
				STATE_TEMPS_RESTANT_PREP := 	STATE_TEMPS_PREPARATION - PRM_TPS_SEGMENT[1] -
													TIME_TO_INT(TIMER_SEGMENT[2].ET / 1000);

			2,3:
				STATE_TEMPS_RESTANT_PREP :=	STATE_TEMPS_RESTANT_PREP;
		END_CASE

		STATE_TEMPS_RESTANT_CLOT := 	STATE_TEMPS_CLOTURE;
		STATE_Temps_Phase 		       := 	INT_TO_TIME(STATE_TEMPS_RESTANT_PREP) * 1000;

	7:
		STATE_Segment 	:= 	3;
		STATE_TEMPS_SEGMENT := TIMER_SEGMENT[3].PT - TIMER_SEGMENT[3].ET;

		CASE PRM_PHASE_PREFFUSION OF
			1:
				STATE_TEMPS_RESTANT_PREP := 	STATE_TEMPS_PREPARATION - PRM_TPS_SEGMENT[1] - PRM_TPS_SEGMENT[2] -
							 						TIME_TO_INT(TIMER_SEGMENT[3].ET / 1000);

			2,3:
				STATE_TEMPS_RESTANT_PREP :=	STATE_TEMPS_RESTANT_PREP;
		END_CASE

		STATE_TEMPS_RESTANT_CLOT := 	STATE_TEMPS_CLOTURE;
		STATE_Temps_Phase 		       := 	INT_TO_TIME(STATE_TEMPS_RESTANT_PREP) * 1000;

	8:
		STATE_Segment	:= 	4;
		STATE_TEMPS_SEGMENT := TIMER_SEGMENT[4].PT - TIMER_SEGMENT[4].ET;

		CASE PRM_PHASE_PREFFUSION OF
			1:
				STATE_TEMPS_RESTANT_PREP := 	STATE_TEMPS_PREPARATION
													- PRM_TPS_SEGMENT[1] - PRM_TPS_SEGMENT[2] - PRM_TPS_SEGMENT[3]
													- TIME_TO_INT(TIMER_SEGMENT[4].ET / 1000);
			2:
				STATE_TEMPS_RESTANT_PREP := 	STATE_TEMPS_PREPARATION
													- TIME_TO_INT(TIMER_SEGMENT[4].ET / 1000);
			3:
				STATE_TEMPS_RESTANT_PREP :=	STATE_TEMPS_RESTANT_PREP;
		END_CASE

		STATE_TEMPS_RESTANT_CLOT := 	STATE_TEMPS_CLOTURE;
		STATE_Temps_Phase 		       := 	INT_TO_TIME(STATE_TEMPS_RESTANT_PREP) * 1000;

	9:
		STATE_Segment	:= 	5;
		STATE_TEMPS_SEGMENT := TIMER_SEGMENT[5].PT - TIMER_SEGMENT[5].ET;

		CASE PRM_PHASE_PREFFUSION OF
			1:
				STATE_TEMPS_RESTANT_PREP := 	STATE_TEMPS_PREPARATION
													- PRM_TPS_SEGMENT[1] - PRM_TPS_SEGMENT[2] - PRM_TPS_SEGMENT[3]
													- PRM_TPS_SEGMENT[4] - TIME_TO_INT(TIMER_SEGMENT[5].ET / 1000);
			2:
				STATE_TEMPS_RESTANT_PREP := 	STATE_TEMPS_PREPARATION
													- PRM_TPS_SEGMENT[4] - TIME_TO_INT(TIMER_SEGMENT[5].ET / 1000);
			3:
				STATE_TEMPS_RESTANT_PREP :=	STATE_TEMPS_RESTANT_PREP;
		END_CASE

		STATE_TEMPS_RESTANT_CLOT := 	STATE_TEMPS_CLOTURE;
		STATE_Temps_Phase 		       := 	INT_TO_TIME(STATE_TEMPS_RESTANT_PREP) * 1000;

	10:
		STATE_Segment 	:= 	6;
		STATE_TEMPS_SEGMENT := TIMER_SEGMENT[6].PT - TIMER_SEGMENT[6].ET;

		CASE PRM_PHASE_PREFFUSION OF
			1:
				STATE_TEMPS_RESTANT_PREP := 	STATE_TEMPS_PREPARATION
													- PRM_TPS_SEGMENT[1] - PRM_TPS_SEGMENT[2] - PRM_TPS_SEGMENT[3]
													- PRM_TPS_SEGMENT[4] - PRM_TPS_SEGMENT[5]
									 				- TIME_TO_INT(TIMER_SEGMENT[6].ET / 1000);
			2:
				STATE_TEMPS_RESTANT_PREP := 	STATE_TEMPS_PREPARATION
													- PRM_TPS_SEGMENT[4] - PRM_TPS_SEGMENT[5]
									 				- TIME_TO_INT(TIMER_SEGMENT[6].ET / 1000);
			3:
				STATE_TEMPS_RESTANT_PREP := 	STATE_TEMPS_PREPARATION
									 				- TIME_TO_INT(TIMER_SEGMENT[6].ET / 1000);
		END_CASE

		STATE_TEMPS_RESTANT_CLOT := 	STATE_TEMPS_CLOTURE;
		STATE_Temps_Phase 		       := 	INT_TO_TIME(STATE_TEMPS_RESTANT_PREP) * 1000;

	11,12:
		STATE_Segment	:=	7;
		STATE_TEMPS_SEGMENT := TIMER_SEGMENT[7].PT - TIMER_SEGMENT[7].ET;

		CASE PRM_PHASE_PREFFUSION OF
			1:
				STATE_TEMPS_RESTANT_PREP := 	STATE_TEMPS_PREPARATION
													- PRM_TPS_SEGMENT[1] - PRM_TPS_SEGMENT[2] - PRM_TPS_SEGMENT[3]
													- PRM_TPS_SEGMENT[4] - PRM_TPS_SEGMENT[5]
													- PRM_TPS_SEGMENT[6] - TIME_TO_INT(TIMER_SEGMENT[7].ET / 1000);
			2:
				STATE_TEMPS_RESTANT_PREP := 	STATE_TEMPS_PREPARATION
													- PRM_TPS_SEGMENT[4] - PRM_TPS_SEGMENT[5]
													- PRM_TPS_SEGMENT[6] - TIME_TO_INT(TIMER_SEGMENT[7].ET / 1000);
			3:
				STATE_TEMPS_RESTANT_PREP := 	STATE_TEMPS_PREPARATION
													- PRM_TPS_SEGMENT[6] - TIME_TO_INT(TIMER_SEGMENT[7].ET / 1000);
		END_CASE

		STATE_Temps_Phase 		       := 	INT_TO_TIME(STATE_TEMPS_RESTANT_PREP) * 1000;
		STATE_TEMPS_RESTANT_CLOT := 	STATE_TEMPS_CLOTURE;

	13:
		STATE_Segment 	:=	8;	(*Phase d'évaporation*)
		STATE_TEMPS_SEGMENT := TIMER_SEGMENT[8].PT - TIMER_SEGMENT[8].ET; (*représente le temps max de dépôt*)
		IF PRM_RATE > 0 THEN
			STATE_TEMPS_RESTANT_DEPOT :=	REAL_TO_INT(((PRM_Thickness*1000) - I_THICKNESS) / PRM_Rate);
		END_IF
		STATE_TEMPS_SEGMENT := T#0ms;
		STATE_Temps_Phase 		       := 	T#0ms;

	14:
		STATE_Segment	:=	9;

		STATE_TEMPS_SEGMENT := TIMER_SEGMENT[9].PT - TIMER_SEGMENT[9].ET;
		STATE_TEMPS_RESTANT_DEPOT := 	0;
		STATE_TEMPS_RESTANT_PREP 	:=	0;
		STATE_TEMPS_RESTANT_CLOT 	:=	STATE_TEMPS_CLOTURE - TIME_TO_INT(TIMER_SEGMENT[9].ET / 1000);

		STATE_Temps_phase		       := 	INT_TO_TIME(STATE_TEMPS_RESTANT_CLOT) * 1000;

	15:
		STATE_Segment	:=	10;
		STATE_TEMPS_SEGMENT := TIMER_SEGMENT[10].PT - TIMER_SEGMENT[10].ET;
		STATE_TEMPS_RESTANT_DEPOT := 	0;
		STATE_TEMPS_RESTANT_PREP 	:=	0;
		STATE_TEMPS_RESTANT_CLOT 	:=	STATE_TEMPS_CLOTURE - PRM_TPS_SEGMENT[9] - TIME_TO_INT(TIMER_SEGMENT[9].ET / 1000);
		STATE_Temps_Phase 		       := 	INT_TO_TIME(STATE_TEMPS_RESTANT_CLOT) * 1000;
	ELSE
		STATE_TEMPS_SEGMENT := T#0ms;
		STATE_Segment	:= 	0;
		STATE_Temps_Phase 		       := 	T#0ms;

END_CASE

(*Calcul de la puissance à appliquer pendant la phase de préfusion*)
IF NOT (STATE_Segment = 0) AND NOT (STATE_Segment = 8) THEN
		IF (STATE_segment = 1) THEN
			VAR_Pi 		:= 	0.0;
		ELSIF (STATE_segment = 9) THEN
			VAR_Pi		:=	MEM_POWER ;
		ELSE
			VAR_Pi		:=	MEM_POWER;  (*PRM_PWR_SEGMENT[STATE_Segment - 1]*)
		END_IF
		VAR_Pf 			:=	PRM_PWR_SEGMENT[STATE_Segment];
		VAR_Time 		:=	TIME_TO_REAL(TIMER_SEGMENT[STATE_Segment].ET) / 1000;
		VAR_Tseg 		:=	PRM_TPS_SEGMENT[STATE_SEGMENT] ;
		IF VAR_Tseg > 0 THEN
			OUT_Power 		:=	(((VAR_Pf - VAR_Pi)/VAR_Tseg)	* VAR_Time) + VAR_Pi;
		ELSE
			OUT_Power 		:= 	VAR_Pf;
		END_IF
END_IF

(*Calcul de la puissance à appliquer pendant la phase d'évaporation*)
IF (STATE_SEGMENT = 8) AND TIMER_Prise_Controle.Q AND NOT PRM_PFixe THEN
		OUT_Power 		:=	I_Power;		(*Application de la consigne du controleur de dépôt*)
ELSIF (STATE_SEGMENT = 8) AND PRM_PFixe THEN
		OUT_Power 		:=	PRM_PWR_SEGMENT[8];		(*Application de la consigne du controleur de dépôt*)
END_IF
IF OP_MARCHE.Etape.0 AND NOT MANUAL OR
	(OP_Marche.Etape.1 AND NOT (PRM_NCR = VAR_Mem_Creuset)) THEN	(*RAZ de la puissance si on utilise pas le même creuset*)
		OUT_POWER	:=	0.0;
		RQ_marche_HT	:=	FALSE;
		RQ_marche_FIL	:=	FALSE;
END_IF

(*Etat de l'évaporation*)
STATE_PREP_OK	:= 	OP_MARCHE.Etape.12;
STATE_EVAP 		:= 	OP_MARCHE.Etape.13;
STATE_CLOT_OK 	:= 	OP_MARCHE.OK OR OP_MARCHE.AR;
STATE_PREFU 		:= 	(STATE_Segment >= 1) AND (STATE_Segment < 8);
STATE_IDLE			:= 	(STATE_Segment = 9) OR (STATE_Segment = 10);
STATE_END_DEPOT_PFIXE	:=	OP_MARCHE.Etape.13 AND (I_THICKNESS >= PRM_Thickness) AND PRM_PFIXE;


FM_ETAPE3_MARCHE(CLK:=OP_MARCHE.Etape.3);
IF FM_ETAPE3_MARCHE.Q THEN
	CONS_HT:=	PRM_HT;
END_IF

(*Gestion de la mémorisation des creusets*)
IF OP_MARCHE.etape.3 THEN
	VAR_Mem_Creuset := PRM_NCR;
END_IF
RQ_Ref_mesure 	:= 	NOT OP_MARCHE.Etape.0 OR OP_STOP.etape.1 OR OP_STOP.etape.2 OR OP_STOP.etape.3;
RQ_Ref_source	:=	NOT OP_MARCHE.Etape.0 OR OP_STOP.etape.1 OR OP_STOP.etape.2 OR OP_STOP.etape.3;

(*marche balayage*)
IF	OP_Marche.Etape.17 THEN
	RQ_marche_SWEEP	:=	TRUE;
ELSIF (OP_Marche.Etape.0 AND OP_Stop.Etape.0) OR OP_STOP.Etape.4 OR RESET OR MANUAL THEN
	RQ_marche_SWEEP	:=	FALSE;
END_IF

(* marche HT *)
IF	OP_Marche.Etape.3 THEN
	RQ_marche_HT 	:= TRUE;
ELSIF (Op_marche.Etape.0 AND OP_stop.Etape.0) OR OP_STOP.Etape.3 THEN
	RQ_marche_HT 	:= FALSE;
END_IF

(* Marche filament*)
IF	OP_Marche.Etape.4 THEN
	RQ_marche_FIL 	:= TRUE;
ELSIF (Op_marche.Etape.0 AND OP_stop.Etape.0) OR OP_STOP.Etape.2 THEN
	RQ_marche_FIL 	:= FALSE;
END_IF

(*Changement de creuset*)
IF OP_Marche.Etape.1 THEN
	RQ_Switch_Crucible := TRUE;
ELSIF (OP_Marche.Etape.0 AND OP_Stop.Etape.0) OR OP_Marche.Etape.17 OR OP_STOP.Etape.4 THEN
	RQ_Switch_Crucible := FALSE;
END_IF

IF OP_MARCHE.Etape.1 THEN
	CONS_NBAL := PRM_NBAL ;
	CONS_NCR := PRM_NCR;
END_IF


(*
IF (Op_marche.Etape.0 AND OP_stop.Etape.0 AND NOT MANUAL) OR OP_STOP.Etape.2 THEN
	CONS_NBAL := 0;
END_IF
*)
(*Seuillage Pmax*)
IF (OUT_POWER >= PRM_PMAX) THEN
	OUT_POWER := PRM_PMAX;
	FLAG_PMAX := TRUE;				(*Flag pour puissance max atteinte*)
ELSE
	FLAG_PMAX := FALSE;
END_IF

(*
IF (OUT_POWER > (PRM_PMAX * 1.05)) THEN
	IF OUT_Power <= 95 THEN
		OUT_Power := PRM_PMAX * 1.05;
	ELSE
		OUT_Power := PRM_PMAX;
	END_IF
	FLAG_PMAX := TRUE;				(*Flag pour puissance max atteinte*)
ELSE
	FLAG_PMAX := FALSE;
END_IF
*)

(*
(*Demande d'ouverture du cache source*)
TIMER_RETARD_FCACHE(
		IN:= VAR_RETARD_FERM_CACHE,
		PT:= REAL_TO_TIME(PRM_RETARD_FERM_CACHE*1000)
		);
VAR_RETARD_FERM_CACHE := FALSE;
TIMER_RETARD_OCACHE(
		IN:= NOT (OP_MARCHE.Etape.5 OR OP_MARCHE.Etape.6 OR OP_MARCHE.Etape.7 OR OP_MARCHE.Etape.8 OR
			OP_MARCHE.Etape.9 OR OP_MARCHE.Etape.10 OR OP_MARCHE.Etape.11 OR OP_MARCHE.Etape.12 OR
			OP_MARCHE.Etape.13) ,
		PT:= REAL_TO_TIME(PRM_REOUV_CACHE*1000),
		);
RQ_Ouv_Cache_source := OP_MARCHE.Etape.13 OR TIMER_RETARD_FCACHE.Q OR (TIMER_RETARD_OCACHE.Q AND
		NOT (PRM_REOUV_CACHE = 0));
*)
RQ_Ouv_Cache_source := OP_MARCHE.Etape.13 AND (I_OUV_CACHE_SOURCE OR PRM_PFixe);

(*Défaut du quartz qui contrôle la vitesse de dépôt*)
DEF_QZ_CTRL_RATE.CONDITION :=  OP_Marche.Etape.13 AND I_DEF_QZ_CTRL_RATE AND NOT I_TIME_POWER;
DEF_QZ_CTRL_RATE.DELAY := T#60s;
DEF_QZ_CTRL_RATE();

(*Défaut de refroidissement*)
DEF_REF.CONDITION := NOT OP_MARCHE.Etape.0 AND (NOT I_ref_mesure_ok OR NOT I_ref_source_ok);
DEF_REF.DELAY := T#5s;
DEF_REF();


(*Défaut de puissance max atteinte*)
DEF_Pmax.CONDITION:= FLAG_PMAX;
DEF_Pmax();

(*Seuillage Pmin pendant la phase de dépôt et d'ajustement vitesse en fin de préfusion*)
IF (OUT_Power <= PRM_PMIN) AND (STATE_Segment = 8) AND (PRM_PMIN > 0) THEN
	OUT_Power:= PRM_PMIN;
	FLAG_PMIN := TRUE;
ELSE
	FLAG_PMIN := FALSE;
END_IF

(*Demande de marche du contrôleur*)
TIMER_Start_Controleur.IN		:=	OP_Marche.Etape.13;
TIMER_Start_Controleur.PT		:=	T#1s;
TIMER_Start_Controleur();
OUT_Start_Controleur	:=	OP_Marche.Etape.13(*TIMER_Start_Controleur.Q*);

(*RAZ consigne vitesse pour affichage sur XTC si puissance fixe*)
IF NOT OP_Marche.AR AND PRM_PFixe THEN
	PRM_Rate	:=	0;
END_IF

(*Défaut de puissance min atteinte*)
DEF_Pmin.CONDITION := FLAG_PMIN AND (op_marche.Etape.13 OR STATE_PREFU);
DEF_Pmin();


(*Surveillance du temps de dépôt théorique à ne pas dépasser*)
(*si le temps théorique est > au temps min alors on ajoute le pourcentage pour le temps d'enveloppe*)
IF (STATE_TEMPS_DEPOT > PRM_TPS_MIN_SURV_DEPOT) AND NOT PRM_PFIXE THEN
	DEF_TEMPS_MAX.DELAY	:=	REAL_TO_TIME(INT_TO_REAL(STATE_TEMPS_DEPOT) * ((100+PRM_FACTEUR_TEMPS_DEPOT)/100)*1000);
ELSIF PRM_PFIXE THEN
	DEF_TEMPS_MAX.DELAY	:=	REAL_TO_TIME(UINT_TO_REAL(PRM_TPS_Max_PFixe)*1000);
(*si le temps théorique  est < au temps min alors on ajoute le temps min pour le temps d'enveloppe*)
ELSE
	DEF_TEMPS_MAX.DELAY	:=	REAL_TO_TIME((INT_TO_REAL(STATE_TEMPS_DEPOT) + PRM_TPS_MIN_SURV_DEPOT)*1000);
END_IF


(*Defaut dépassement du temps max de dépôt*)
DEF_TEMPS_MAX(
				CONDITION:= OP_Marche.Etape.13  AND ( DEF_TEMPS_MAX.DELAY > T#0ms),
				);


STATE_AR := (OP_MARCHE.Etape.0 AND OP_STOP.Etape.0) OR OP_STOP.OK;

(*Reset demandes*)
CO_Modif	:=	FALSE;
END_ACTION

ACTION PRL:
OP_MARCHE.IdXML		:=	'0';
OP_MARCHE.TagXML	:=	1;

OP_STOP.IdXML		:=	'0';
OP_STOP.TagXML		:=	2;

DEF_QZ_CTRL_RATE.IDXML := '14';
DEF_QZ_CTRL_RATE.TagXML := 8;

DEF_PMAX.IdXML	:=	'14';
DEF_PMAX.TagXML	:=	10;

DEF_PMIN.IdXML := '14';
DEF_Pmin.TagXML := 12;

DEF_TEMPS_MAX.IdXML := '14';
DEF_TEMPS_MAX.TagXML  := 11;

DEF_REF.IdXML := '14';
DEF_REF.TagXML:= 28;
END_ACTION

END_FUNCTION_BLOCK

// ---- POUs/Composant/BLOCK_ACTUATOR.TcPOU
FUNCTION_BLOCK BLOCK_ACTUATOR

(* Gestion d'un actionneur monostable ou bistable avec ou sans retour d'état *)

(****************historique des versions*****************************)

(* Version 1-0 - SP - VERSION INIITIALE 6844 DP650 N35*)
(* Version 2-0 - HG - Adaptation pour journal des évènements externe - 24/06/2011*)
(*************************************************************************)


VAR_INPUT
	I_PARAM_SYSTEM_OK:			BOOL;											(*paramétrage système ok*)
(*paramètre standard*)
	RESET:   					BOOL; 											(*Condition RAZ actionneur*)
	MANUAL:  					BOOL; 											(*Mode manuel*)
(*entrée externe*)
	IN_OFF:						BOOL; (* ~ (OPC : 1 : available for OPC-clients) *)		(*E.TOR actionneur au repos*)
	IN_ON:						BOOL; (* ~ (OPC : 1 : available for OPC-clients) *)		(*E.TOR actionneur actif*)
(*défaut du bloc*)
	DEF_On:  					PRCDEF; 									(*01 - Défaut d'ouverture de la vanne de transfert*)
	DEF_Off:   					PRCDEF;	 									(*02 - Défaut de fermeture de la vanne de transfert*)
	DEF_Sensor:  				PRCDEF; 									(*03 - Défaut d'incohérence des capteurs de la vanne de transfert*)
	DEF_On_Imposs:				PRCDEF;										(*04 - Défaut d'activation non autorisé en mode automatique*)
	DEF_Off_Imposs:				PRCDEF;										(*05 - Défaut de désactivation non autorisée en mode automatique*)
	DEF_Off_auto:				PRCDEF;										(*06 - Défaut de désactivation automatique*)

(*parametre de pilotage en entrée*)
	CO_On:   					BOOL; 				(*Ordre mode automatique activation*)
	CO_Off:  					BOOL;				(*Ordre mode automatique désactivation*)
	EN_On_INT:   				BOOL:=TRUE;			(*Condition d'autorisation d'activation donnée par le bloc qui instancie le bloc actuator*)
	EN_Off_INT:  				BOOL:=TRUE;			(*Condition d'autorisation de désactivation donnée par le bloc qui instacie le bloc actuator*)
	EN_On_EXT:					BOOL:=TRUE;			(*condition d'autorisation d'activation externe*)
	EN_Off_EXT:					BOOL:=TRUE;			(*condition d'autorisation de desactivation externe*)
END_VAR

VAR_INPUT PERSISTENT
(*parametre de configuration constructeur*)
(*les parametres suivants dépendent de la configuration de la machine*)
	CONF_Type_Actuator: 		USINT:=0;										(*définit le type d'actionneur
																				*0 = monostable
																				1 = bistable *)

	CONF_EN_On:					USINT:=0;				(*définit la réaction du système en cas de perte des conditions d'autorisation d'activation EN_On
														 0 = désactivation automatique  en cas de perte des conditions d'autorisation d'activation uniquement en manuel
														 1 = désactivation automatique en cas de perte des conditions d'autorisation d'activation en auto et en manuel
														 2 = Pas de déscativation automatique*)
	CONF_DI_Off:   				BOOL:=FALSE;									(*option de presence d'un capteur desactivation*)
	CONF_DI_On:  				BOOL:=FALSE;									(*option de presence d'un capteur activation ok*)
	CONF_No_Safety_Auto:		BOOL:=FALSE;									(*option de desactivation des conditions d'autorisation en mode automatique*)
	CONF_Tim_Valid_On:  		TIME; 											(*Temps validation actionneur on*)
	CONF_Tim_Valid_Off:   		TIME; 											(*Temps validation actionneur off *)

	(*Entité*)
	IsComponent:		BOOL;			(*entité : composant*)
	IdXML:				STRING;			(*nom entité : identifiant pour recherche dans dico*)
	TagXML:				UINT;			(*nom entité : identifiant pour recherche dans dico*)
	IdParent:			STRING;			(*MNEMO de l'appelant*)
	MNEMO:				STRING;			(*MNEMO de l'entité*)
END_VAR

VAR_OUTPUT
	OUT_On:					BOOL;	(* ~ (OPC : 1 : available for OPC-clients) *)		(*SORTIE TOR ACTIVATION*)
	OUT_Off:				BOOL; 	(* ~ (OPC : 1 : available for OPC-clients) *)		(*SORTIE TOR DESACTIVATION*)
	STATE_On:	   			BOOL; 	(* ~ (OPC : 1 : available for OPC-clients) *)		(*Indicateur activation ok*)
	STATE_Off:  			BOOL; 	(* ~ (OPC : 1 : available for OPC-clients) *)		(*Indicateur désactivation ok*)
	STATE_Nok:				BOOL;	(* ~ (OPC : 1 : available for OPC-clients) *)		(*Indicateur défaut sur l'actionneur*)
	AUTOR_On_IHM:			BOOL; 	(* ~ (OPC : 1 : available for OPC-clients) *)		(*etat activation autorisée depuis la supervision*)
	AUTOR_Off_IHM:			BOOL; 	(* ~ (OPC : 1 : available for OPC-clients) *)		(*etat désactivation autorisée depuis la supervision*)
	AUTOR_On_PLC:			BOOL;											(*etat activation autorisée depuis l'automate*)
	AUTOR_Off_PLC:			BOOL;											(*etat désactivation autorisée depuis l'automate*)
END_VAR


VAR
	TIMER_Valid_On:			TON;
	TIMER_Valid_Off:		TON;

	M_On:  						BOOL; 	(* ~ (OPC : 1 : available for OPC-clients) *)		(*Ordre mode manuel activation ou activation/desactivation si la vanne est monostable*)
	M_Off:   					BOOL; 	(* ~ (OPC : 1 : available for OPC-clients) *)		(*Ordre mode manuel désactivation*)
	RCP_M_On:   				BOOL;
	RCP_M_Off:  				BOOL;
	VAR_On:						BOOL;											(*variable intermédiaire avant affectation de la sortie OUT_On *)
	VAR_Off:					BOOL;											(*Variable intermédiaire avant affectation de la sortie OUT_Off *)

	VAR_CPT:					BLOCK_CPT_APP;
END_VAR

VAR_EXTERNAL
	MANUAL_SAFETY_OFF:	BOOL;												(*desactive les sécurités en mode manuel*)
END_VAR

(* Réception des ordres en mode manuel*)
RCP_M_On 			:=	M_On;
RCP_M_Off			:=	M_Off;
(*Autorisation*)
AUTOR_On_IHM		:= 	MANUAL AND ((EN_On_INT AND EN_On_EXT)
						OR MANUAL_SAFETY_OFF) AND NOT RESET AND NOT VAR_On;
AUTOR_Off_IHM		:= 	MANUAL AND ((EN_Off_INT AND EN_Off_EXT)  OR
						MANUAL_SAFETY_OFF) AND NOT RESET AND NOT VAR_Off;
AUTOR_On_PLC		:=	NOT MANUAL AND ((EN_On_INT AND EN_On_EXT)
						OR CONF_No_Safety_Auto) AND NOT RESET;
AUTOR_Off_PLC		:= 	NOT MANUAL AND ((EN_Off_INT AND EN_Off_EXT)
						OR CONF_No_Safety_Auto) AND NOT RESET;

(*defaut activation impossible en mode automatique*)
DEF_On_Imposs.CONDITION:=	(CO_On AND NOT AUTOR_On_PLC) AND NOT RESET AND NOT MANUAL;
DEF_On_Imposs.DELAY := T#0ms;
DEF_On_Imposs();
(*Defaut désactivation impossible en mode automatique*)
DEF_Off_Imposs.CONDITION:=	(CO_Off AND NOT AUTOR_Off_PLC AND (CONF_TYPE_ACTUATOR=1)) OR
							(NOT CO_On AND VAR_On  AND NOT AUTOR_Off_PLC AND (CONF_TYPE_ACTUATOR=0))
							AND NOT RESET AND NOT MANUAL;
DEF_Off_Imposs.DELAY := T#0ms;
DEF_Off_Imposs();
(*defaut desactivation automatique*)
DEF_Off_Auto.CONDITION :=   (NOT EN_On_INT OR NOT EN_On_EXT) AND  VAR_On AND ((CONF_En_ON=1)
							OR ((CONF_EN_On=0) AND MANUAL)) AND NOT RESET;
DEF_Off_auto.DELAY:=T#0ms;
DEF_Off_Auto();

(*gestion des sorties*)
IF 		(RCP_M_On AND AUTOR_On_IHM) OR
		(CO_On AND AUTOR_On_PLC) THEN
				VAR_On		:= 	TRUE;
				VAR_Off		:= 	FALSE;
ELSIF 	(RCP_M_Off AND AUTOR_Off_IHM AND (CONF_Type_Actuator=1)) OR
		(RCP_M_On AND AUTOR_Off_IHM AND (CONF_Type_Actuator=0)) OR
	    	(CO_Off AND AUTOR_Off_PLC AND (CONF_Type_Actuator=1)) OR
		(NOT CO_On AND AUTOR_Off_PLC AND (CONF_Type_Actuator=0))
		OR (RESET AND (CONF_Type_Actuator=0)) OR
		DEF_Off_Auto.DEF THEN
				VAR_On		:=	FALSE;
				VAR_Off		:=	TRUE;
ELSIF 	RESET AND (CONF_Type_Actuator=1)   THEN
				VAR_On		:= 	FALSE;
				VAR_Off		:=	FALSE;
END_IF;



OUT_On		:=	VAR_On;
OUT_OFF		:=	VAR_Off AND (CONF_type_Actuator = 1);

(*indicateur actionneur activé STATE_ON*)
TIMER_Valid_On.IN	:=	((NOT IN_OFF AND CONF_DI_Off AND NOT CONF_DI_On) OR
						(VAR_ON AND NOT CONF_DI_On AND NOT CONF_DI_Off) OR
						(IN_ON AND CONF_DI_On) AND NOT DEF_SENSOR.DEF);
TIMER_Valid_On(PT:=CONF_Tim_Valid_On);
STATE_ON			:=	TIMER_Valid_On.Q;
(*indicateur actionneur activé STATE_OFF*)
TIMER_Valid_Off.IN	:=	((NOT IN_ON AND CONF_DI_On AND NOT CONF_DI_Off) OR
						(VAR_OFF AND NOT CONF_DI_On AND NOT CONF_DI_Off) OR
						(IN_OFF AND CONF_DI_Off) AND NOT DEF_SENSOR.DEF);
TIMER_Valid_Off(PT:=CONF_Tim_Valid_Off);
STATE_Off			:=	TIMER_Valid_Off.Q;

(*indicateur STATE_NOK*)
STATE_Nok			:=	DEF_ON.DEF OR DEF_Off.DEF OR DEF_Sensor.DEF OR DEF_On_Imposs.DEF OR DEF_Off_Imposs.DEF OR DEF_Off_auto.DEF;

(*défaut d'activation*)
DEF_On.Condition	:= 	VAR_On AND NOT STATE_On AND (CONF_DI_Off OR CONF_DI_On) AND NOT RESET;
DEF_On();
(*défaut désactivation*)
DEF_Off.Condition	:= 	VAR_Off AND NOT STATE_Off AND (CONF_DI_Off OR CONF_DI_On) AND NOT RESET;
DEF_Off();
(*défaut capteur*)
DEF_Sensor.Condition	:= 	IN_On AND IN_Off AND CONF_DI_Off AND CONF_DI_On AND NOT RESET;
DEF_Sensor();

(*gestion compteur*)
VAR_CPT(I_On:= STATE_On);

(* Reset des ordres *)
IF M_On AND RCP_M_On THEN
	M_On 	:= FALSE;
END_IF;
IF M_Off AND RCP_M_Off THEN
	M_Off		 := FALSE;
END_IF;

END_FUNCTION_BLOCK

// ---- POUs/Composant/EVAP/BLOCK_CANON_ST10.TcPOU
FUNCTION_BLOCK BLOCK_CANON_ST10

(* Gestion d'une source Telemark ST-10 *)

(****************historique des versions*****************************)

(* Version 0 - GV - 01/2015  - affaire 8866 EVA760 n°12 *)

(*************************************************************************)

VAR_INPUT
	DOOR:						BOOL;		(*porte fermée*)
	VAC:						BOOL;		(*sécurité vide*)
	WATER:						BOOL;		(*refroidissement canon ok*)
	MANUAL:						BOOL;		(*demande mode manuel*)
	I_CR_OK:					BOOL;		(*Positionnement creuset ok*)
	RESET:						BOOL;		(*reset*)

	AI_UHV:						ANALOG_INPUT;
	AI_IEM:						ANALOG_INPUT;
	AI_FIL:						ANALOG_INPUT;
	IN_UHVQ			AT%I*:		INT;			(* Entrée analogique Haute Tension *)
	IN_IEMQ			AT%I*:		INT;			(* Entrée analogique courant d'émission *)
	IN_FILQ			AT%I*:		INT;			(* Entrée analogique courant filament *)

	IN_HV_OK		AT%I*:		BOOL;		(* Entrée TOR Haute Tension prête *)
	IN_HV_ON		AT%I*:		BOOL;		(* Entrée TOR Haute tension ON *)
	IN_SRC_ON		AT%I*:		BOOL;		(* Entrée TOR Source ON *)

	HV:							BLOCK_ACTUATOR;
	SRC:						BLOCK_ACTUATOR;

	I_TENSION:					REAL;		(*consigne de tension (kV) appliquée en mode automatique*)
	PRM_TENSION:				REAL;		(*Consigne de tension (kV) appliquée en mode manuel*)
	I_COURANT:					REAL;		(*consigne de courant (%) appliquée en mode automatique*)
	PRM_COURANT:				REAL;		(*Consigne de courant (%) appliquée en mode manuel*)
	CO_HV:						BOOL;		(*Commande externe de marche de la Haute Tension en automatique*)
	CO_SRC:						BOOL;		(*commande de marche de la source en automatique*)

END_VAR

VAR_INPUT PERSISTENT
	(*Entité*)
	IsComponent:		BOOL;			(*entité : composant*)
	IdXML:				STRING;			(*nom entité : identifiant pour recherche dans dico*)
	TagXML:				UINT;			(*nom entité : identifiant pour recherche dans dico*)
	IdParent:			STRING;			(*MNEMO de l'appelant*)
	MNEMO:				STRING;			(*MNEMO de l'entité*)
END_VAR

VAR_OUTPUT
	OUT_HV				AT%Q*:		BOOL;			(*Pilotage de la haute tension*)
	OUT_SRC				AT%Q*:		BOOL;			(*Pilotage de la source*)
	OUT_QUHV			AT%Q*:		INT;			(*Sortie analogique de la consigne tension (max 10kV) *)
	OUT_QIEM			AT%Q*:		INT;			(*Sortie analogique de la consigne courant emission (max 1000mA)*)
	OUT_ITLCK_VAC	 	AT%Q*:		BOOL;			(*Interlock de vide Haute Tension*)
	OUT_ITLCK_HVAC		AT%Q*:		BOOL;			(*Interlock de vide Source*)
	OUT_ITLCK_WAT		AT%Q*:		BOOL;			(*Interlock eau source*)
	AO_QUHV:						ANALOG_OUTPUT;
	AO_QIEM:						ANALOG_OUTPUT;

